	REGION 7 - Handle handshake
	    #iqUDT_HandShakeDownstreamSlip.RTS := #iqUDT_HandShakeUpstream.RTS;
	    #iqUDT_HandShakeUpstream.RTR := #iqUDT_HandShakeDownstreamSlip.RTR;
	    #iqUDT_HandShakeDownstreamSlip.TIP := #iqUDT_HandShakeUpstream.TIP;
	    #iqUDT_HandShakeDownstreamSlip.ResetEnergySave := #iqUDT_HandShakeUpstream.ResetEnergySave;
	    #iqUDT_HandShakeUpstream.CascadeStartUp := #iqUDT_HandShakeDownstreamSlip.CascadeStartUp;
	    #iqUDT_HandShakeDownstreamSlip.ReqStop := #iqUDT_HandShakeUpstream.ReqStop;
	    #iqUDT_HandShakeDownstreamSlip.DownstreamDisplacement := #iqUDT_ConveyorInterfaceDownstream.Displacement;
	END_REGION

END_FUNCTION_BLOCK

FUNCTION_BLOCK "FB_SoftVersion"
TITLE = FB_SoftVersion
{ S7_Optimized_Access := 'TRUE' }
AUTHOR : MHSE
FAMILY : GeneralSystemFunctions
VERSION : 3.0
// ATTRIBUTES
// AUTO_NUMBER = True
// BLOCK_NUMBER = 28
// END_ATTRIBUTES
//Function block to get the program checksums.
   VAR_INPUT
      is_ActualDateTime { ExternalAccessible := 'False'; ExternalVisible := 'False'; ExternalWritable := 'False'} : String;   // Actual date and time
   END_VAR

   VAR_OUTPUT
      qs_SoftVersion { ExternalAccessible := 'False'; ExternalVisible := 'False'; ExternalWritable := 'False'} : String[8];   // Software version
      qa_StandardCRC { ExternalAccessible := 'False'; ExternalVisible := 'False'; ExternalWritable := 'False'} : Array[0..7] of Byte;   // Standard program checksum output
      qa_SafetyCRC { ExternalAccessible := 'False'; ExternalVisible := 'False'; ExternalWritable := 'False'} : Array[0..7] of Byte;   // Safety program checksum output
   END_VAR

   VAR
      sFB_GetChecksum_Safety {InstructionName := 'GetChecksum'; LibVersion := '1.0'; ExternalAccessible := 'False'; ExternalVisible := 'False'; ExternalWritable := 'False'; S7_SetPoint := 'False'} : GetChecksum;   // Safety checksum read block
      sFB_GetChecksum_Standard {InstructionName := 'GetChecksum'; LibVersion := '1.0'; ExternalAccessible := 'False'; ExternalVisible := 'False'; ExternalWritable := 'False'; S7_SetPoint := 'False'} : GetChecksum;   // Standard checksum read block
   END_VAR
   VAR RETAIN
      sa_StandardCRC { ExternalAccessible := 'False'; ExternalVisible := 'False'; ExternalWritable := 'False'} : Array[0..7] of Byte;   // Standard program checksum
      sa_SafetyCRC { ExternalAccessible := 'False'; ExternalVisible := 'False'; ExternalWritable := 'False'} : Array[0..7] of Byte;   // Safety program checksum
   END_VAR
   VAR
      sa_NewStandardCRC { ExternalAccessible := 'False'; ExternalVisible := 'False'; ExternalWritable := 'False'} : Array[0..7] of Byte;   // New standard program checksum
      sa_NewSafetyCRC { ExternalAccessible := 'False'; ExternalVisible := 'False'; ExternalWritable := 'False'} : Array[0..7] of Byte;   // New safety program checksum
   END_VAR
   VAR RETAIN
      ss_Date { ExternalAccessible := 'False'; ExternalVisible := 'False'; ExternalWritable := 'False'} : String[8];   // Date charater string
   END_VAR

   VAR_TEMP
      ta_StandardCRC : Struct   // GetChecksum
         tx_Done : Bool;   // GetChecksum - Done
         tx_Busy : Bool;   // GetChecksum - Busy
         tx_Error : Bool;   // GetChecksum - Error
         tw_Status : Word;   // GetChecksum - Status
      END_STRUCT;
      ta_SafetyCRC : Struct   // GetChecksum
         tx_Done : Bool;   // GetChecksum - Done
         tx_Busy : Bool;   // GetChecksum - Busy
         tx_Error : Bool;   // GetChecksum - Error
         tw_Status : Word;   // GetChecksum - Status
      END_STRUCT;
      tx_CRCValid : Bool;   // Checksums valid
   END_VAR


BEGIN
	(*
	----------------------------------------------------------------------------------------

	Version history:
	Date        | Version   | Author        | Remark
	----------------------------------------------------------------------------------------
	24/05/2019  | 0.1       | K.Pokorski    | first release MHS TIA 15.1
	14/06/2019  | 0.2       | A.Nowak       | Replacement of instruction if for direct write into variable - Region 2
	24/07/2019  | 2.0       | L.Klar        | 2.0 MHS library release TIA 15.1
	27/08/2019  | 2.2       | K.Pokorski    | Comments adjusted
	12/11/2019  | 3.0       | P.Majka       | 3.0 MHS library release TIA 15.1
	21/02/2023  | 4.0       | F.Baten       | 4.0 Release TIA 17.5
	*)

	REGION 1 - Standard and safety program checksums

	    // Scope - 1 - Standard program CRC
	    #sFB_GetChecksum_Standard(Scope := 1,
	                              Done => #ta_StandardCRC.tx_Done,
	                              Busy => #ta_StandardCRC.tx_Busy,
	                              Error => #ta_StandardCRC.tx_Error,
	                              Status => #ta_StandardCRC.tw_Status,
	                              Checksum := #sa_NewStandardCRC);

	    // Scope - 2 - Safety program CRC
	    #sFB_GetChecksum_Safety(Scope := 2,
	                            Done => #ta_SafetyCRC.tx_Done,
	                            Busy => #ta_SafetyCRC.tx_Busy,
	                            Error => #ta_SafetyCRC.tx_Error,
	                            Status => #ta_SafetyCRC.tw_Status,
	                            Checksum := #sa_NewSafetyCRC);

	END_REGION

	REGION 2 - Checksums comparison

	    #tx_CRCValid := (#sa_NewStandardCRC = #sa_StandardCRC)
	    AND (#sa_SafetyCRC = #sa_NewSafetyCRC);

	END_REGION

	REGION 3 - New software version

	    // Separate the year, mounth and day from actual date and time and connect it to one string
	    IF (NOT #tx_CRCValid)                                           // Checksums not valid
	    THEN

	        #ss_Date := CONCAT(IN1 := MID(IN := #is_ActualDateTime,
	                                                         L := 4,
	                                                         P := 1),

	                           IN2 := MID(IN := #is_ActualDateTime,
	                                      L := 2,
	                                      P := 6),

	                           IN3 := MID(IN := #is_ActualDateTime,
	                                      L := 2,
	                                      P := 9));

	        // Standard progrm checksum update
	        #sa_StandardCRC := #sa_NewStandardCRC;

	        // Safety program checksum update
	        #sa_SafetyCRC := #sa_NewSafetyCRC;

	    END_IF;

	END_REGION

	REGION 4 - Write outputs

	    // New program date
	    #qs_SoftVersion := #ss_Date;

	    // Actual standard program checksum
	    #qa_StandardCRC := #sa_StandardCRC;

	    // Actual safety program checksum
	    #qa_SafetyCRC := #sa_SafetyCRC;

	END_REGION
END_FUNCTION_BLOCK

FUNCTION_BLOCK "FB_VfdNORDPPO4"
TITLE = Control block for NORD VFD with PPO4
{ S7_Optimized_Access := 'TRUE' }
AUTHOR : MHS
VERSION : 0.1
// ATTRIBUTES
// AUTO_NUMBER = True
// BLOCK_NUMBER = 235
// END_ATTRIBUTES
   VAR_INPUT
      iUDT_VFDConfig { ExternalAccessible := 'False'; ExternalVisible := 'False'; ExternalWritable := 'False'} : "UDT_VfdConfiguration";   // Configuration structure
      iUDT_VFDInputs { ExternalAccessible := 'False'; ExternalVisible := 'False'; ExternalWritable := 'False'} : "UDT_VfdNordPI";   // VFD inputs structure
      iUDT_MotorData { ExternalAccessible := 'False'; ExternalVisible := 'False'; ExternalWritable := 'False'} : "UDT_MotorData";   // Motor data structure
      ix_24vOk { ExternalAccessible := 'False'; ExternalVisible := 'False'; ExternalWritable := 'False'} : Bool;   // TRUE when 24VDC is healthy
      ix_400vOk { ExternalAccessible := 'False'; ExternalVisible := 'False'; ExternalWritable := 'False'} : Bool;   // TRUE when 400VAC is healthy
      ix_QuickStopDisable { ExternalAccessible := 'False'; ExternalVisible := 'False'; ExternalWritable := 'False'} : Bool := FALSE;   // TRUE when Motor can turn, False = Quick stop
      ix_SimulationModeActive { ExternalAccessible := 'False'; ExternalVisible := 'False'; ExternalWritable := 'False'} : Bool;   // TRUE when Simulation mode active
   END_VAR

   VAR_OUTPUT
      qUDT_HMIStatus { ExternalAccessible := 'False'; ExternalVisible := 'False'; ExternalWritable := 'False'} : "UDT_VfdStatus";   // HMI status structure
      qUDT_VFDOutputs { ExternalAccessible := 'False'; ExternalVisible := 'False'; ExternalWritable := 'False'} : "UDT_VfdNordPO";   // VFD outputs structure
      qUDT_commisioning { ExternalAccessible := 'False'; ExternalVisible := 'False'; ExternalWritable := 'False'} : "UDT_CommisioningNord";
   END_VAR

   VAR_IN_OUT
      iqUDT_ConveyorInterface : "UDT_ConveyorInterface";   // Conveyor interface structure
      iqUDT_VFDStatistics : "UDT_VfdStatistics";   // Satistics structure
      iqx_StartCommissioning { ExternalAccessible := 'False'; ExternalVisible := 'False'; ExternalWritable := 'False'} : Bool;   // TRUE when Start auto-commissioning
   END_VAR

   VAR
      sFB_TimerOnOffDelayCheck24V { ExternalAccessible := 'False'; ExternalVisible := 'False'; ExternalWritable := 'False'; S7_SetPoint := 'False'} : "FB_TimerOnOffDelay";   // MHS "TimerOnOffDelay" - to delay time for VFD 24V contactor
      sFB_TimerOnOffDelayCheck400V { ExternalAccessible := 'False'; ExternalVisible := 'False'; ExternalWritable := 'False'; S7_SetPoint := 'False'} : "FB_TimerOnOffDelay";   // MHS "TimerOnOffDelay" - to delay time for VFD 400V contactor
      sFB_TimerOnOffDelayVFDReset { ExternalAccessible := 'False'; ExternalVisible := 'False'; ExternalWritable := 'False'; S7_SetPoint := 'False'} : "FB_TimerOnOffDelay";   // MHS "TimerOnOffDelay" - to extend VFD reset
      sFB_TimerOnOffDelayVFDRunningFeedbackError { ExternalAccessible := 'False'; ExternalVisible := 'False'; ExternalWritable := 'False'; S7_SetPoint := 'False'} : "FB_TimerOnOffDelay";   // MHS "TimerOnOffDelay" - to delay time for VFDRunningFeedback error
      sFB_VfdNORDCommissiong { ExternalAccessible := 'False'; ExternalVisible := 'False'; ExternalWritable := 'False'; S7_SetPoint := 'False'} : "FB_VfdNORDCommissioning";   // FB to commissiong NORD drive
      sUDT_Status { ExternalAccessible := 'False'; ExternalVisible := 'False'; ExternalWritable := 'False'; S7_SetPoint := 'False'} : "UDT_VfdStatus";   // Detailed VFD status overview
      sUDT_PNDevice { ExternalAccessible := 'False'; ExternalVisible := 'False'; ExternalWritable := 'False'; S7_SetPoint := 'False'} : "UDT_PNDevice";   // PN device info structure
      sa_PNPortsStatus { ExternalAccessible := 'False'; ExternalVisible := 'False'; ExternalWritable := 'False'} : Array[1..8] of Bool;   // TRUE when specific port has an error
      sp_VFDTelegram { ExternalAccessible := 'False'; ExternalVisible := 'False'; ExternalWritable := 'False'} : HW_ANY;   // Free telegram's HW_ID
      sv_VFDGeoStruct {InstructionName := 'GEOADDR'; LibVersion := '1.0'; ExternalAccessible := 'False'; ExternalVisible := 'False'; ExternalWritable := 'False'; S7_SetPoint := 'False'} : GEOADDR;   //  Geo structure indicate to telegram
      sR_TRIG_PNSlaveNotOnline {InstructionName := 'R_TRIG'; LibVersion := '1.0'; ExternalAccessible := 'False'; ExternalVisible := 'False'; ExternalWritable := 'False'; S7_SetPoint := 'False'} : R_TRIG;   // Rising edge for trigger Profinet slave not online statistics
      sR_TRIG_PNSlaveError {InstructionName := 'R_TRIG'; LibVersion := '1.0'; ExternalAccessible := 'False'; ExternalVisible := 'False'; ExternalWritable := 'False'; S7_SetPoint := 'False'} : R_TRIG;   // Rising edge for trigger Profinet slave error statistics
      sR_TRIG_VFDInternalError {InstructionName := 'R_TRIG'; LibVersion := '1.0'; ExternalAccessible := 'False'; ExternalVisible := 'False'; ExternalWritable := 'False'; S7_SetPoint := 'False'} : R_TRIG;   // Rising edge for trigger Internal VFD Error statistics
      sR_TRIG_Running {InstructionName := 'R_TRIG'; LibVersion := '1.0'; ExternalAccessible := 'False'; ExternalVisible := 'False'; ExternalWritable := 'False'; S7_SetPoint := 'False'} : R_TRIG;   // Rising edge for starting of the running signal
      sF_TRIG_RunFwd {InstructionName := 'F_TRIG'; LibVersion := '1.0'; ExternalAccessible := 'False'; ExternalVisible := 'False'; ExternalWritable := 'False'; S7_SetPoint := 'False'} : F_TRIG;   // Falling edge for run forward signal
      sF_TRIG_RunRvs {InstructionName := 'F_TRIG'; LibVersion := '1.0'; ExternalAccessible := 'False'; ExternalVisible := 'False'; ExternalWritable := 'False'; S7_SetPoint := 'False'} : F_TRIG;   // Falling edge for run reverse signal
      sr_RPMActual { ExternalAccessible := 'False'; ExternalVisible := 'False'; ExternalWritable := 'False'} : Real;   // Drive RPM feedback
      sr_RPMSetpoint { ExternalAccessible := 'False'; ExternalVisible := 'False'; ExternalWritable := 'False'} : Real;   // Actual speed setpoint [rpm]
      sr_ReferenceFrequency { ExternalAccessible := 'False'; ExternalVisible := 'False'; ExternalWritable := 'False'} : Real;   // Frequency of the reference RPM in [Hz]
      sdi_LastRampTimeUp { ExternalAccessible := 'False'; ExternalVisible := 'False'; ExternalWritable := 'False'} : UDInt;   // Last cycle ramp down time
      sdi_LastRampTimeDown { ExternalAccessible := 'False'; ExternalVisible := 'False'; ExternalWritable := 'False'} : UDInt;   // Last cycle ramp up time
      si_ActualRamp { ExternalAccessible := 'False'; ExternalVisible := 'False'; ExternalWritable := 'False'} : UInt;   // Actual ramp value
      si_ActualRampUpTime { ExternalAccessible := 'False'; ExternalVisible := 'False'; ExternalWritable := 'False'} : UInt;   // Actual ramp up time
      si_ActualRampDownTime { ExternalAccessible := 'False'; ExternalVisible := 'False'; ExternalWritable := 'False'} : UInt;   // Actual ramp down time
      si_HWAdress { ExternalAccessible := 'False'; ExternalVisible := 'False'; ExternalWritable := 'False'} : Int;
      si_ActualSpeed { ExternalAccessible := 'False'; ExternalVisible := 'False'; ExternalWritable := 'False'} : Int;   // Actual speed in [mm/sec]
      si_Log2GeoReturn { ExternalAccessible := 'False'; ExternalVisible := 'False'; ExternalWritable := 'False'} : Int;   // Log2Geo function return
      si_Geo2LogReturn { ExternalAccessible := 'False'; ExternalVisible := 'False'; ExternalWritable := 'False'} : Int;   // Geo2Log function return
      sx_ConfigurationError { ExternalAccessible := 'False'; ExternalVisible := 'False'; ExternalWritable := 'False'} : Bool;   // Commissioning: configuration error
      sx_PNDeviceHealthy { ExternalAccessible := 'False'; ExternalVisible := 'False'; ExternalWritable := 'False'} : Bool;   // Profinet device is online and error free
      sx_HardwareAvailable { ExternalAccessible := 'False'; ExternalVisible := 'False'; ExternalWritable := 'False'} : Bool;   // Power and communication to drive are ok
      sx_VfdAvailable { ExternalAccessible := 'False'; ExternalVisible := 'False'; ExternalWritable := 'False'} : Bool;   // Hardware of VFD is ok and no communication error with movikit
      sx_24vOk { ExternalAccessible := 'False'; ExternalVisible := 'False'; ExternalWritable := 'False'} : Bool;   // 24VDC is healthy
      sx_400vOk { ExternalAccessible := 'False'; ExternalVisible := 'False'; ExternalWritable := 'False'} : Bool;   // 400VAC is healthy
      sx_ErrorActive { ExternalAccessible := 'False'; ExternalVisible := 'False'; ExternalWritable := 'False'} : Bool;   // Block has an error
      sx_EnableOperation { ExternalAccessible := 'False'; ExternalVisible := 'False'; ExternalWritable := 'False'} : Bool;   // Enable operation signal
      sx_RunVFDReverse { ExternalAccessible := 'False'; ExternalVisible := 'False'; ExternalWritable := 'False'} : Bool;   // Start VFD backward
      sx_RunVFDForward { ExternalAccessible := 'False'; ExternalVisible := 'False'; ExternalWritable := 'False'} : Bool;   // Start VFD forward
      sx_SpeedSetpointReached { ExternalAccessible := 'False'; ExternalVisible := 'False'; ExternalWritable := 'False'} : Bool;   // Motor is running at requested speed
      sx_VFDStopping { ExternalAccessible := 'False'; ExternalVisible := 'False'; ExternalWritable := 'False'} : Bool;   // VFD Stopping
      sx_VFDNotReadyError { ExternalAccessible := 'False'; ExternalVisible := 'False'; ExternalWritable := 'False'} : Bool;   // Temporary Error need to be implemented in the status
   END_VAR

   VAR CONSTANT
      cr_MaximumValueSpeedWord : Real := 16384.0;   // Maximum value of speed actual value
      cr_MaximumValueRampWord : Real := 32767.0;   // Maximum value of ramp setpoint ( corresponds to 20Sec)
      cr_MaximumFrequency : Real := 16384.0;   // Maximum value of frequency setpoint (corresponds to P105 Maximum Frequency)
      cudi_DefaultRampDownTime : UDInt := 20000;   // VFD ramp down default time [ms]
      cudi_DefaultRampUpTime : UDInt := 20000;   // VFD ramp up default time [ms]
      ci_VFDArea : UInt := 1;   // Area ID of IO Profinet devices
      ci_SubmoduleHWType : UInt := 5;   // Submodule HW_type number
      ci_TelegramSlot : UInt := 0;   // PPO4 telegram slot
      ci_TelegramSubslot : UInt := 1;   // PPO4 telegram subslot
      ci_NumberOfProfinetPorts : Int := 2;   // Number of Profinet ports in device
   END_VAR


BEGIN
	(*
	----------------------------------------------------------------------------------------

	Version history:
	Date        | Version   | Author        | Remark
	----------------------------------------------------------------------------------------
	25/01/2020  | 0.1       | S.Theocharis  | Initial version TIA 15.1
	28/04/2022  | 0.2       | K. Pokorski   | NORD Commissioning interface change
	09/05/2022  | 0.3       | M. Pluskota   | Reference speed changed to nominal speed for actual speed calculation
	12/05/2022  | 0.4       | M. Pluskota   | Ramp equation adjustet for nord drives
	04/06/2022  | 0.5       | M. Pluskota   | Aded a if statment to not exceed the max value of the ramp value
	                                        | Error decoding changed now the error is shown as ErrorCode.SubErrorCodee
	12/07/2022  | 0.6       | M. Pluskota   | Ramp equation bug fix
	29/07/2022  | 0.7       | M. Piela      | Add hardware ok to the profinet checking
	21/02/2023  | 4.0       | F.Baten       | 4.0 Release TIA 17.5
	*)


	REGION 1 - Get Device Profinet information

	    "FC_GetDevicePN"(is_PNDeviceName := #iUDT_VFDConfig.VFDPNDeviceName,
	                     ix_SimulationModeActive := #ix_SimulationModeActive,
	                     iqUDT_PND := #sUDT_PNDevice);


	    "FC_GetPNPortStatus"(ii_NumberOfPorts := #ci_NumberOfProfinetPorts,
	                         iUDT_DevicePNInfo := #sUDT_PNDevice,
	                         qa_PortFault => #sa_PNPortsStatus);

	END_REGION

	REGION 2 - Reset errors

	    IF #iqUDT_ConveyorInterface.InternalErrorReset OR (NOT #iqUDT_ConveyorInterface.HardwareOk AND #sUDT_Status.PNSlaveNotonline)   // Reser errors when Reset is given
	    THEN

	        #sUDT_Status.PNSlaveNotonline := FALSE;
	        #sUDT_Status.PNSlaveError := FALSE;
	        #sUDT_Status.InternalError := FALSE;
	        #sUDT_Status.VFDRunningFeedbackError := FALSE;
	        #sUDT_Status.PNSlaveWarning := FALSE;

	    END_IF;


	    // Create  extended pulse for VFD Reset
	    #sFB_TimerOnOffDelayVFDReset(iudi_OnDelayTime := 0,
	                                 iudi_OffDelayTime := 200,
	                                 ix_SignalToDelay := #iqUDT_ConveyorInterface.InternalErrorReset,
	                                 ix_Enable := TRUE);

	END_REGION

	REGION 3 - Hardware checks
	    // Hardware will only be available after the delay, so the device has time for the initialisation
	    #sFB_TimerOnOffDelayCheck24V(iudi_OnDelayTime := 2000,
	                                 iudi_OffDelayTime := 0,
	                                 ix_SignalToDelay := #ix_24vOk
	    );

	    #sx_24vOk := #sFB_TimerOnOffDelayCheck24V.qx_DelayedSignal;

	    #sFB_TimerOnOffDelayCheck400V(iudi_OnDelayTime := 2000,
	                                  ix_SignalToDelay := #ix_400vOk);

	    #sx_400vOk := #sFB_TimerOnOffDelayCheck400V.qx_DelayedSignal;

	    // Check if PN device is online
	    IF NOT "DB_ProfinetDiagnostic".ProfinetNetworks[#sUDT_PNDevice.PNNetworknumber].DeviceStatus[#sUDT_PNDevice.PNDeviceNumber].DeviceState.Exist
	        AND NOT #ix_SimulationModeActive
	        AND #sx_24vOk
	        AND #iqUDT_ConveyorInterface.HardwareOk
	    THEN
	        #sUDT_Status.PNSlaveNotonline := TRUE;

	    END_IF;

	    // Check if PN ports are healthy
	    IF #sa_PNPortsStatus[1] XOR #sa_PNPortsStatus[2] THEN
	        #sUDT_Status.PNSlaveWarning := TRUE;
	    END_IF;


	    // Check if PN device has an error
	    IF "DB_ProfinetDiagnostic".ProfinetNetworks[#sUDT_PNDevice.PNNetworknumber].DeviceStatus[#sUDT_PNDevice.PNDeviceNumber].DeviceState.Error
	        AND NOT #ix_SimulationModeActive
	        AND #sx_24vOk
	        AND NOT #sUDT_Status.PNSlaveWarning
	        AND #iqUDT_ConveyorInterface.HardwareOk
	    THEN
	        #sUDT_Status.PNSlaveError := TRUE;
	    END_IF;

	    // Set bit when PN device is healthy (online and no error)
	    #sx_PNDeviceHealthy := NOT #sUDT_Status.PNSlaveNotonline
	    AND NOT #sUDT_Status.PNSlaveError
	    AND #sUDT_PNDevice.PNDeviceFound
	    AND #sx_24vOk;

	    // Set hardware available bit when all conditions are met
	    #sx_HardwareAvailable := (#sx_24vOk
	    AND #sx_PNDeviceHealthy)
	    OR #ix_SimulationModeActive;


	    // VFD is ready for operation if hardware ok
	    #sx_VfdAvailable := #sx_HardwareAvailable;

	    //VFD not ready error . Temporary
	    #sx_VFDNotReadyError := #sx_HardwareAvailable
	    AND NOT #iUDT_VFDInputs.ZSW.ReadyToStart
	    AND #iUDT_VFDInputs.ZSW.EmergencyStop
	    OR NOT #iUDT_VFDInputs.ZSW.BusControlActive;




	END_REGION

	REGION 4 - Check errors and warnings

	    // Check if the VFD has a warning
	    #sUDT_Status.InternalWarning := #iUDT_VFDInputs.ZSW.WarningActive;

	    // Copy warning code to status DB when warning active
	    IF #sUDT_Status.InternalWarning
	    THEN

	        #sUDT_Status.ErrorCode := #iUDT_VFDInputs.FaultCode / 10; // AST check the value of warning
	        #sUDT_Status.SubErrorCode := #iUDT_VFDInputs.FaultCode MOD 10;

	    END_IF;

	    // Check if the VFD has an error
	    #sUDT_Status.InternalError := #iUDT_VFDInputs.ZSW.Fault; // AND NOT #sx_StartMeasuring;

	    // Copy error code to status DB when error active
	    IF #sUDT_Status.InternalError
	    THEN

	        #sUDT_Status.ErrorCode := #iUDT_VFDInputs.FaultCode / 10; // AST check the value of warning
	        #sUDT_Status.SubErrorCode := #iUDT_VFDInputs.FaultCode MOD 10;

	    END_IF;

	    // Reset error code if warning and error not available
	    IF (NOT #sUDT_Status.InternalWarning
	        AND NOT #sUDT_Status.InternalError)
	    THEN

	        #sUDT_Status.ErrorCode := 0;
	        #sUDT_Status.SubErrorCode := 0;
	    END_IF;

	END_REGION

	REGION 5 - Check if configuration is ok for commissioning purposes

	    IF #iUDT_VFDConfig.WheelEndPerimeter > 0.0                                         // If perimeter of wheel at the end of gear is greater than 0
	        AND #iUDT_VFDConfig.GearRatio > 0.0                                            // and gear ratio is greater than 0
	        AND #iUDT_VFDConfig.ReferenceRPM > 0.0                                         // and maximum speed is greater than 0
	        AND #iUDT_VFDConfig.VFDRampUpTime > 0                                          // and ramp up time is greater than 0
	        AND #iUDT_VFDConfig.VFDRampDownTime > 0                                        // and ramp down time is greater than zero
	        AND #iUDT_VFDConfig.VFDStartupTime > 0.0                                       // and startup time is greater then zero
	        //  AND MOTOR NOMINAL SPEED IS >0  the reference speed is invalid for NORD drives
	        AND #cudi_DefaultRampUpTime > #iUDT_VFDConfig.VFDRampUpTime                     // and ramp up time is not greater than default ramp up time
	        AND #cudi_DefaultRampDownTime > #iUDT_VFDConfig.VFDRampDownTime                 // and ramp down time is not greater than default ramp down time
	        // need to know if the FI receives a percentage of a default ramp or value in ms , depending to that the configuration validation code will change

	        AND (#sUDT_PNDevice.PNDeviceFound                                              // and device not found in PN structure
	        OR #ix_SimulationModeActive)                                                    // or simulation mode is active
	    THEN
	        #sx_ConfigurationError := FALSE;                                                // Reset configuration error
	    ELSE
	        #sx_ConfigurationError := TRUE;                                                 // Set configuration error
	    END_IF;
	    #qUDT_commisioning.CommissionError := #sx_ConfigurationError;

	END_REGION

	REGION 6 - Speed handling

	    //Calculate actual speed value in rpm
	    // #sr_RPMActual := ((INT_TO_REAL(#i_UDT_VFDInputs.ActualSpeed) / #cr_MaximumValueSpeedWord) * INT_TO_REAL(#i_UDT_MotorData.NominalSpeed));

	    //#sr_RPMActual := ((INT_TO_REAL(#i_UDT_VFDInputs.ActualSpeed) / #cr_MaximumValueSpeedWord) * (#i_UDT_MotorData.NominalSpeed));
	    #sr_RPMActual := ((INT_TO_REAL(#iUDT_VFDInputs.ActualSpeed) / #cr_MaximumFrequency) * (#iUDT_VFDConfig.ReferenceRPM));
	    // Calculate actual speed in mm/s
	    #si_ActualSpeed := REAL_TO_INT((#sr_RPMActual / #iUDT_VFDConfig.GearRatio) * ((#iUDT_VFDConfig.WheelEndPerimeter) / 60.0));


	    //change the i_UDT_VFDInput.Actualspeed to RPM

	    // Reversal actual speed
	    IF #iUDT_VFDConfig.DirectionReversal THEN

	        #si_ActualSpeed := #si_ActualSpeed * -1;

	    END_IF;

	    // Calculate actual speed setpoint in rpm
	    #sr_RPMSetpoint := ((DINT_TO_REAL(INT_TO_DINT(#iqUDT_ConveyorInterface.SpeedSetpoint) * 60)) / #iUDT_VFDConfig.WheelEndPerimeter) * #iUDT_VFDConfig.GearRatio;

	    // Check if speed setpoint is reached
	    #sx_SpeedSetpointReached := (ABS(#si_ActualSpeed) >= (#iqUDT_ConveyorInterface.SpeedSetpoint - #iUDT_VFDConfig.SpeedSetpointWindow))
	    AND (ABS(#si_ActualSpeed) <= (#iqUDT_ConveyorInterface.SpeedSetpoint + #iUDT_VFDConfig.SpeedSetpointWindow));


	END_REGION

	REGION 7 - Prepare output data VFD

	    REGION 7.1 - Set speed setpoint in forward and reverse directory

	        // If motor stopped and Run forward is requested and interlock forward is active, the speed setpoint is loaded to run forward.
	        //  IF (#i_UDT_VFDInputs.ActualSpeed = 0) AND #iq_UDT_ConveyorInterface.RunFwd AND #i_UDT_VFDConfig.InterlockFwd
	        IF #iqUDT_ConveyorInterface.RunFwd AND #iUDT_VFDConfig.InterlockFwd
	        THEN
	            #sx_RunVFDForward := TRUE;
	            #sx_RunVFDReverse := FALSE;
	        END_IF;

	        // If motor stopped and Run reverse is requested and interlock reverse is active, the speed setpoint is loaded to run reverse.
	        IF (#iUDT_VFDInputs.ActualSpeed = 0) AND #iqUDT_ConveyorInterface.RunRvs AND #iUDT_VFDConfig.InterlockRvs
	        THEN
	            #sx_RunVFDReverse := TRUE;
	            #sx_RunVFDForward := FALSE;
	        END_IF;

	    END_REGION

	    REGION 7.2 - Stopping

	        // Create trigger when direction signal falling
	        #sF_TRIG_RunFwd(CLK := #iqUDT_ConveyorInterface.RunFwd);
	        #sF_TRIG_RunRvs(CLK := #iqUDT_ConveyorInterface.RunRvs);

	        // When no run signal is given the VFD should stop
	        IF NOT #iqUDT_ConveyorInterface.RunRvs AND NOT #iqUDT_ConveyorInterface.RunFwd
	            OR (#iqUDT_ConveyorInterface.RunRvs AND #iqUDT_ConveyorInterface.RunFwd)
	            OR #sF_TRIG_RunRvs.Q
	            OR #sF_TRIG_RunFwd.Q

	        THEN
	            #sx_RunVFDReverse := FALSE;
	            #sx_RunVFDForward := FALSE;
	        END_IF;

	        IF NOT #sx_RunVFDReverse AND NOT #sx_RunVFDForward AND (#iUDT_VFDInputs.ActualSpeed <> 0)
	        THEN
	            #sx_VFDStopping := TRUE;
	        ELSE
	            #sx_VFDStopping := FALSE;
	        END_IF;

	    END_REGION

	    REGION 7.3 - Check for enable operation signal

	        #sx_EnableOperation := #sx_VfdAvailable
	        AND #sx_400vOk
	        AND NOT #sx_ConfigurationError
	        AND (#sx_RunVFDForward OR #sx_RunVFDReverse); // add communication error

	    END_REGION

	    REGION 7.4 - Write acceleration and deceleration value to drive

	        //Detect is VFD is ramping up
	        IF ABS(#sr_RPMSetpoint) > ABS(#sr_RPMActual)
	            AND NOT #sx_SpeedSetpointReached
	            AND #iUDT_VFDInputs.ZSW.OperationEnabled
	            AND (#sx_RunVFDForward OR #sx_RunVFDReverse)
	        THEN
	            // Calculate the ramp up time if the vfd configuration is changed durning process or the vfd starts from speed 0
	            IF #sdi_LastRampTimeUp <> #iUDT_VFDConfig.VFDRampUpTime THEN
	                #si_ActualRamp := REAL_TO_UINT(UDINT_TO_REAL(#iUDT_VFDConfig.VFDRampUpTime) / UDINT_TO_REAL(#cudi_DefaultRampUpTime) * #cr_MaximumValueRampWord / (#sr_RPMSetpoint / #iUDT_VFDConfig.ReferenceRPM));
	                #si_ActualRampUpTime := #si_ActualRamp;
	            ELSE
	                #si_ActualRamp := #si_ActualRampUpTime;
	            END_IF;
	            #sdi_LastRampTimeUp := #iUDT_VFDConfig.VFDRampUpTime;
	        ELSE
	            // Calculate the ramp down time if the actual speed is greater than 0 and the configuration has changed durning process
	            // or the VFD perform the first deceleration

	            IF #si_ActualSpeed <> 0 THEN
	                IF #sdi_LastRampTimeDown <> #iUDT_VFDConfig.VFDRampDownTime
	                THEN
	                    #si_ActualRamp := REAL_TO_UINT(UDINT_TO_REAL(#iUDT_VFDConfig.VFDRampDownTime) / UDINT_TO_REAL(#cudi_DefaultRampDownTime) * #cr_MaximumValueRampWord / (#sr_RPMSetpoint / #iUDT_VFDConfig.ReferenceRPM));
	                    #si_ActualRampDownTime := #si_ActualRamp;

	                ELSE
	                    #si_ActualRamp := #si_ActualRampDownTime;
	                END_IF;
	                #sdi_LastRampTimeDown := #iUDT_VFDConfig.VFDRampDownTime;
	            ELSE
	                #sdi_LastRampTimeDown := 0;
	                #sdi_LastRampTimeUp := 0;
	            END_IF;

	        END_IF;

	        // If the ramp value exceeds the maximum value, then the maximum value is sent to the VFD
	        IF UINT_TO_REAL(#si_ActualRamp) > #cr_MaximumValueRampWord
	        THEN
	            #qUDT_VFDOutputs.RampTimeSetPoint := REAL_TO_INT(#cr_MaximumValueRampWord);
	        ELSE
	            #qUDT_VFDOutputs.RampTimeSetPoint := REAL_TO_INT(UINT_TO_REAL(#si_ActualRamp));
	        END_IF;


	    END_REGION
	END_REGION

	REGION 8 - Auto Commmissioning

	    REGION 8.1 Initialize
	        IF #iqx_StartCommissioning THEN

	            //Caclulate theoretical reference Hz. Necessary for NORD drives cause the setpoint is given at Hz
	            //Variation of motor slip from 50Hz to reference Hz is not taken into account. That means there will always be a variantion between Setpoint and actual speed
	            #sr_ReferenceFrequency := (#iUDT_VFDConfig.ReferenceRPM / 1500) * 50; //1500 for 4 pole motor

	            // Get hardware adres of "SK-TU4-PNS~Head" submodule
	            #si_Log2GeoReturn := LOG2GEO(LADDR := "DB_ProfinetDiagnostic".ProfinetNetworks[#sUDT_PNDevice.PNNetworknumber].DeviceStatus[#sUDT_PNDevice.PNDeviceNumber].DeviceState.HW_ID, GEOADDR := #sv_VFDGeoStruct);       // "LOG2GEO" to get profinet network number
	            #sv_VFDGeoStruct.AREA := #ci_VFDArea;                                                                                                                                                                               // Set IO Profinet devices area ID
	            #sv_VFDGeoStruct.HWTYPE := #ci_SubmoduleHWType;                                                                                                                                                                     // Set submodule HW_type number
	            #sv_VFDGeoStruct.STATION := INT_TO_UINT(#sUDT_PNDevice.PNDeviceNumber);                                                                                                                                            // Set device's profinet number
	            #sv_VFDGeoStruct.SLOT := #ci_TelegramSlot;                                                                                                                                                                          // Set free telegram slot
	            #sv_VFDGeoStruct.SUBSLOT := #ci_TelegramSubslot;                                                                                                                                                                    // Set free telegram subslot

	            #si_Geo2LogReturn := GEO2LOG(GEOADDR := #sv_VFDGeoStruct, LADDR => #sp_VFDTelegram);                                                                                                                              // "GEO2LOG" to get free telegram's HW_ID

	        END_IF;

	    END_REGION

	    REGION 8.2 Run - auto commissioning

	        #sFB_VfdNORDCommissiong(ix_VFDReadyToRun := #sx_400vOk AND #iUDT_VFDInputs.ZSW.EmergencyStop AND NOT #iUDT_VFDInputs.ZSW.Fault,
	                                qx_24VCommissioningDone => #sFB_VfdNORDCommissiong.qx_24VCommissioningDone,
	                                iqx_Enable := #iqx_StartCommissioning,
	                                ir_ReferenceFrequency := #sr_ReferenceFrequency,
	                                ihw_HardwareID := #sp_VFDTelegram,
	                                iudt_MotorData := #iUDT_MotorData,
	                                qi_HWAdress => #qUDT_commisioning.HWAdress,
	                                qx_Busy => #sFB_VfdNORDCommissiong.qx_Busy,
	                                qx_Done => #sFB_VfdNORDCommissiong.qx_Done,
	                                qx_Error => #sFB_VfdNORDCommissiong.qx_Error);

	    END_REGION

	END_REGION

	REGION 9 - Write outputs to VFD

	    REGION 9.1 - Write control word 1

	        #qUDT_VFDOutputs.STW.ReadyForOperation := #sx_RunVFDReverse OR #sx_RunVFDForward;
	        #qUDT_VFDOutputs.STW.DisableVoltage := TRUE;
	        #qUDT_VFDOutputs.STW.EmergencyStop := #ix_QuickStopDisable;
	        #qUDT_VFDOutputs.STW.EnableOperation := TRUE;
	        #qUDT_VFDOutputs.STW.EnablePulsles := TRUE;
	        #qUDT_VFDOutputs.STW.EnableRamp := TRUE;
	        #qUDT_VFDOutputs.STW.EnableSetpoint := TRUE;
	        #qUDT_VFDOutputs.STW.Acknowledge := #sFB_TimerOnOffDelayVFDReset.qx_DelayedSignal;
	        #qUDT_VFDOutputs.STW."StartFunction408.11" := FALSE;
	        #qUDT_VFDOutputs.STW."StartFunction408.12" := FALSE;
	        #qUDT_VFDOutputs.STW.ControlDataValid := TRUE;
	        #qUDT_VFDOutputs.STW.RotationRightOn := TRUE; //direction reversal via the speed setpoint
	        #qUDT_VFDOutputs.STW.RotationLeftOn := FALSE;
	        #qUDT_VFDOutputs.STW.Reserved := FALSE;
	        #qUDT_VFDOutputs.STW.ParameterSetBit0 := FALSE; //Parameter set 1
	        #qUDT_VFDOutputs.STW.ParameterSetBit1 := FALSE; //Parameter set 1

	        IF (NOT #sx_VfdAvailable OR NOT #sx_400vOk) //AND NOT #sx_StartMeasuring
	        THEN
	            #qUDT_VFDOutputs.STW.ReadyForOperation := FALSE;
	            #qUDT_VFDOutputs.STW.EmergencyStop := FALSE;
	            #qUDT_VFDOutputs.STW.EnableSetpoint := FALSE;
	            #qUDT_VFDOutputs.STW."StartFunction408.11" := FALSE;
	            #qUDT_VFDOutputs.STW."StartFunction408.12" := FALSE;
	        END_IF;
	    END_REGION

	    REGION 9.2 - Write speed setpoint to drive

	        // Calculate normalized speed setpoint
	        #qUDT_VFDOutputs.FrequencySetPoint := REAL_TO_INT((#sr_RPMSetpoint / #iUDT_VFDConfig.ReferenceRPM) * #cr_MaximumFrequency);

	        IF #qUDT_VFDOutputs.FrequencySetPoint > #cr_MaximumFrequency
	        THEN
	            #qUDT_VFDOutputs.FrequencySetPoint := REAL_TO_INT(#cr_MaximumFrequency);
	        END_IF;

	        // The conveyor stopped and may now run in reverse direction
	        IF (#sx_RunVFDReverse AND NOT #iUDT_VFDConfig.DirectionReversal)
	            OR (#sx_RunVFDForward AND #iUDT_VFDConfig.DirectionReversal)
	        THEN
	            #qUDT_VFDOutputs.FrequencySetPoint := #qUDT_VFDOutputs.FrequencySetPoint * -1;
	        END_IF;

	        // Clear speed setpoint when no run request or above direction request or is configuration error
	        IF (NOT #sx_RunVFDForward AND NOT #sx_RunVFDReverse)
	            OR #sx_ConfigurationError
	        THEN
	            #qUDT_VFDOutputs.FrequencySetPoint := 0;
	        END_IF;

	    END_REGION

	END_REGION

	REGION 10 - Check if motor is running

	    //The motor should start running after specific time. If not the VFDRunningFeedback error occured
	    #sFB_TimerOnOffDelayVFDRunningFeedbackError(iudi_OnDelayTime := #iUDT_VFDConfig.VFDStartupTime,
	                                                ix_SignalToDelay := #sx_EnableOperation AND NOT (#si_ActualSpeed <> 0));

	    IF #sFB_TimerOnOffDelayVFDRunningFeedbackError.qx_DelayedSignal THEN

	        #sUDT_Status.VFDRunningFeedbackError := TRUE;

	    END_IF;



	END_REGION

	REGION 11 - Copy signals to interface DB and to status output UDT

	    // Create internal error status
	    #sx_ErrorActive := #sUDT_Status.PNSlaveNotonline
	    OR #sUDT_Status.VFDRunningFeedbackError
	    OR #sUDT_Status.PNSlaveError //Commented out BY AST TO allow run in ring topology v3.12
	    OR #sUDT_Status.InternalError;

	    // Write interface bits - AST Check thoses statuses
	    #iqUDT_ConveyorInterface.VFDRunning := #sx_VfdAvailable AND (#iqUDT_ConveyorInterface.ActualSpeed <> 0 OR #qUDT_VFDOutputs.STW.ReadyForOperation);   // Write true on output Conveyor interface structure if VFD is in operation and motor is turning
	    #iqUDT_ConveyorInterface.VFDatSpeed := #sx_SpeedSetpointReached AND #sx_VfdAvailable AND #si_ActualSpeed <> 0;                                                                                                  // Copy setpoint speed reached state from static to the output conveyor interface structure
	    #iqUDT_ConveyorInterface.InternalWarningVFD := #iUDT_VFDInputs.ZSW.WarningActive;                                                                                                      // Set the internal VFD warning bit if any warning is active
	    #iqUDT_ConveyorInterface.InternalErrorVFD := #sx_ErrorActive;                                                                                                                           // Set the internal VFD error bit if any fault is active
	    #iqUDT_ConveyorInterface.ActualSpeed := #si_ActualSpeed;                                                                                                                                // Copy the calculated value to the output
	    #iqUDT_ConveyorInterface.ConfigurationError := #iqUDT_ConveyorInterface.ConfigurationError OR #sx_ConfigurationError;

	    // Copy error status to output
	    #qUDT_HMIStatus := #sUDT_Status;

	END_REGION

	REGION 12 - Statistic
	    // Create trigger on error and create statistics for profinet slave not online
	    #sR_TRIG_PNSlaveNotOnline(CLK := #sUDT_Status.PNSlaveNotonline);                                        // Detect the rising edge of the error

	    IF #iqUDT_ConveyorInterface.ResetStatistics OR #sUDT_Status.PNSlaveNotonline
	    THEN

	        "FC_Statistics"(ix_Reset := #iqUDT_ConveyorInterface.ResetStatistics,
	                        ix_Activate := #sUDT_Status.PNSlaveNotonline,
	                        ix_RTrigActivate := #sR_TRIG_PNSlaveNotOnline.Q,
	                        iqUDT_Statistics := #iqUDT_VFDStatistics.PNSlaveNotOnline);
	    END_IF;

	    // Create trigger on error and create statistics for profinet slave error
	    #sR_TRIG_PNSlaveError(CLK := #sUDT_Status.PNSlaveError);                                        // Detect the rising edge of the error

	    IF #iqUDT_ConveyorInterface.ResetStatistics OR #sUDT_Status.PNSlaveError
	    THEN

	        "FC_Statistics"(ix_Reset := #iqUDT_ConveyorInterface.ResetStatistics,
	                        ix_Activate := #sUDT_Status.PNSlaveError,
	                        ix_RTrigActivate := #sR_TRIG_PNSlaveError.Q,
	                        iqUDT_Statistics := #iqUDT_VFDStatistics.PNSlaveError);
	    END_IF;

	    // Create trigger on error and create statistics for internal VFD Error
	    #sR_TRIG_VFDInternalError(CLK := #sUDT_Status.InternalError);                                        // Detect the rising edge of the error

	    IF #iqUDT_ConveyorInterface.ResetStatistics OR #sUDT_Status.InternalError
	    THEN

	        "FC_Statistics"(ix_Reset := #iqUDT_ConveyorInterface.ResetStatistics,
	                        ix_Activate := #sUDT_Status.InternalError,
	                        ix_RTrigActivate := #sR_TRIG_VFDInternalError.Q,
	                        iqUDT_Statistics := #iqUDT_VFDStatistics.VFDInternalError);
	    END_IF;

	    // Create trigger on running signal and create statistics for running status
	    #sR_TRIG_Running(CLK := #iqUDT_ConveyorInterface.VFDRunning);                                        // Detect the rising edge of the signal

	    IF #iqUDT_ConveyorInterface.ResetStatistics OR #iqUDT_ConveyorInterface.VFDRunning
	    THEN

	        "FC_Statistics"(ix_Reset := #iqUDT_ConveyorInterface.ResetStatistics,
	                        ix_Activate := #iqUDT_ConveyorInterface.VFDRunning,
	                        ix_RTrigActivate := #sR_TRIG_Running.Q,
	                        iqUDT_Statistics := #iqUDT_VFDStatistics.Running);
	    END_IF;

	END_REGION
END_FUNCTION_BLOCK

FUNCTION_BLOCK "FB_SystemStatistics"
{ S7_Optimized_Access := 'TRUE' }
AUTHOR : MHS
VERSION : 3.0
// ATTRIBUTES
// AUTO_NUMBER = True
// BLOCK_NUMBER = 29
// END_ATTRIBUTES
   VAR_INPUT
      ix_HMIStop { ExternalAccessible := 'False'; ExternalVisible := 'False'; ExternalWritable := 'False'} : Bool;   // HMI stop button one shot signal
      ix_FieldStop { ExternalAccessible := 'False'; ExternalVisible := 'False'; ExternalWritable := 'False'} : Bool;   // Field stop button one shot signal
      ix_BuildingEStop { ExternalAccessible := 'False'; ExternalVisible := 'False'; ExternalWritable := 'False'} : Bool;   // TRUE if bulding emergency stop button is active
      ix_MCPEStop { ExternalAccessible := 'False'; ExternalVisible := 'False'; ExternalWritable := 'False'} : Bool;   // TRUE if MCP emergency stop button is active
      ix_RemotePanelEStop { ExternalAccessible := 'False'; ExternalVisible := 'False'; ExternalWritable := 'False'} : Bool;   // TRUE if Remote Panel emergency stop button is active
   END_VAR

   VAR_IN_OUT
      iqUDT_EquipmentControl : "UDT_EquipmentControl";   // Equipment control structure
      iqUDT_Statistics : "UDT_SystemStatistics";   // Statistics structure
   END_VAR

   VAR
      sR_Trig_HMIStop {InstructionName := 'R_TRIG'; LibVersion := '1.0'; ExternalAccessible := 'False'; ExternalVisible := 'False'; ExternalWritable := 'False'; S7_SetPoint := 'False'} : R_TRIG;   // Rise trigger when a HMI stop is active
      sR_Trig_FieldStop {InstructionName := 'R_TRIG'; LibVersion := '1.0'; ExternalAccessible := 'False'; ExternalVisible := 'False'; ExternalWritable := 'False'; S7_SetPoint := 'False'} : R_TRIG;   // Rise trigger when a field stop is active
      sR_Trig_BuildingEStop {InstructionName := 'R_TRIG'; LibVersion := '1.0'; ExternalAccessible := 'False'; ExternalVisible := 'False'; ExternalWritable := 'False'; S7_SetPoint := 'False'} : R_TRIG;   // Rise trigger when a building emergency stop is active
      sR_Trig_MCPEStop {InstructionName := 'R_TRIG'; LibVersion := '1.0'; ExternalAccessible := 'False'; ExternalVisible := 'False'; ExternalWritable := 'False'; S7_SetPoint := 'False'} : R_TRIG;   // Rise trigger when a MCP emergency stop is active
      sR_Trig_RemotePanelEStop {InstructionName := 'R_TRIG'; LibVersion := '1.0'; ExternalAccessible := 'False'; ExternalVisible := 'False'; ExternalWritable := 'False'; S7_SetPoint := 'False'} : R_TRIG;   // Rise trigger when a remote panel emergency stop is active
      sR_TRIG_AutomaticOn {InstructionName := 'R_TRIG'; LibVersion := '1.0'; ExternalAccessible := 'False'; ExternalVisible := 'False'; ExternalWritable := 'False'; S7_SetPoint := 'False'} : R_TRIG;   // Rise trigger when a automatic mode  is active
      sR_TRIG_DataReset {InstructionName := 'R_TRIG'; LibVersion := '1.0'; ExternalAccessible := 'False'; ExternalVisible := 'False'; ExternalWritable := 'False'; S7_SetPoint := 'False'} : R_TRIG;   // Rise trigger when data reset command is received
      sR_TRIG_Error {InstructionName := 'R_TRIG'; LibVersion := '1.0'; ExternalAccessible := 'False'; ExternalVisible := 'False'; ExternalWritable := 'False'; S7_SetPoint := 'False'} : R_TRIG;   // Rise trigger when  Error occured
      sF_TRIG_Error {InstructionName := 'F_TRIG'; LibVersion := '1.0'; ExternalAccessible := 'False'; ExternalVisible := 'False'; ExternalWritable := 'False'; S7_SetPoint := 'False'} : F_TRIG;   // Fall trigger when  Error is cleared
      sx_HMIStop { ExternalAccessible := 'False'; ExternalVisible := 'False'; ExternalWritable := 'False'} : Bool;   // HMI stop signal
      sx_FieldStop { ExternalAccessible := 'False'; ExternalVisible := 'False'; ExternalWritable := 'False'} : Bool;   // Field stop signal
   END_VAR


BEGIN
	(*
	----------------------------------------------------------------------------------------

	Version history:
	Date        | Version   | Author        | Remark
	----------------------------------------------------------------------------------------
	14/01/2020  | 3.0       | S. Nikodem    | first release MHS TIA 15.1
	22/08/2020  | 3.1       | S. Theocharis | Updated for UPS EMA HMI
	03/08/2021  | 3.2       | M. Roijen     | Bug fix System in error iq_UDT_Statistics
	21/02/2023  | 4.0       | F.Baten       | 4.0 Release TIA 17.5
	*)

	REGION 1 – Triggers

	    // Rise trigger when a HMI stop is active
	    #sR_Trig_HMIStop(CLK := #sx_HMIStop);

	    // Rise trigger when a field stop is active
	    #sR_Trig_FieldStop(CLK := #sx_FieldStop);

	    // Rise trigger when a building emergency stop is active trigger
	    #sR_Trig_BuildingEStop(CLK := #ix_BuildingEStop);

	    // Rise trigger when a MCP emergency stop is active
	    #sR_Trig_MCPEStop(CLK := #ix_MCPEStop);

	    // Rise trigger when a remote panel emergency stop is active
	    #sR_Trig_RemotePanelEStop(CLK := #ix_RemotePanelEStop);

	    // Rise trigger when a Field stop is active
	    #sR_TRIG_AutomaticOn(CLK := #iqUDT_EquipmentControl.Command.AutomaticOn);

	    // Fall trigger when error is cleared (UPS EMA Addition)
	    #sF_TRIG_Error(CLK := #iqUDT_EquipmentControl.Report.Error);

	    //Rise trigger when data reset command is received (UPS EMA Addition)
	    #sR_TRIG_DataReset(CLK := #iqUDT_EquipmentControl.Command.ResetData);

	    //Rise trigger on error
	    #sR_TRIG_Error(CLK := #iqUDT_EquipmentControl.Report.Error);

	END_REGION

	REGION 2 – Sustain input signals

	    // Set HMI stop when input signal and automatic mode are active
	    IF #ix_HMIStop AND #iqUDT_EquipmentControl.Command.AutomaticOn THEN

	        #sx_HMIStop := TRUE;

	    END_IF;

	    // Set Field stop when input signal and automatic mode are active
	    IF #ix_FieldStop AND #iqUDT_EquipmentControl.Command.AutomaticOn THEN

	        #sx_FieldStop := TRUE;

	    END_IF;

	    /// Reset when automatic mode is active
	    IF #sR_TRIG_AutomaticOn.Q THEN

	        #sx_HMIStop := FALSE;
	        #sx_FieldStop := FALSE;

	    END_IF;
	END_REGION

	REGION 3 – Statistics

	    // HMI stop signal statistics
	    IF #sx_HMIStop
	        OR #iqUDT_EquipmentControl.Command.ResetData
	    THEN

	        "FC_Statistics"(ix_Reset := #iqUDT_EquipmentControl.Command.ResetData,
	                        ix_Activate := #sx_HMIStop,
	                        ix_RTrigActivate := #sR_Trig_HMIStop.Q,
	                        iqUDT_Statistics := #iqUDT_Statistics.HMI_Stop);
	    END_IF;

	    // Field stop signal statistics
	    IF #sx_FieldStop
	        OR #iqUDT_EquipmentControl.Command.ResetData
	    THEN

	        "FC_Statistics"(ix_Reset := #iqUDT_EquipmentControl.Command.ResetData,
	                        ix_Activate := #sx_FieldStop,
	                        ix_RTrigActivate := #sR_Trig_FieldStop.Q,
	                        iqUDT_Statistics := #iqUDT_Statistics."Field_Stop");
	    END_IF;

	    // Building emergency stop statistics
	    IF #ix_BuildingEStop
	        OR #iqUDT_EquipmentControl.Command.ResetData
	    THEN

	        "FC_Statistics"(ix_Reset := #iqUDT_EquipmentControl.Command.ResetData,
	                        ix_Activate := #ix_BuildingEStop,
	                        ix_RTrigActivate := #sR_Trig_BuildingEStop.Q,
	                        iqUDT_Statistics := #iqUDT_Statistics."Building_EStop");
	    END_IF;


	    // MCP emergency stop statistics
	    IF #ix_MCPEStop
	        OR #iqUDT_EquipmentControl.Command.ResetData
	    THEN

	        "FC_Statistics"(ix_Reset := #iqUDT_EquipmentControl.Command.ResetData,
	                        ix_Activate := #ix_MCPEStop,
	                        ix_RTrigActivate := #sR_Trig_MCPEStop.Q,
	                        iqUDT_Statistics := #iqUDT_Statistics."MCP_EStop");

	    END_IF;

	    // Remote panel emergency stop statistics
	    IF #ix_RemotePanelEStop
	        OR #iqUDT_EquipmentControl.Command.ResetData
	    THEN

	        "FC_Statistics"(ix_Reset := #iqUDT_EquipmentControl.Command.ResetData,
	                        ix_Activate := #ix_RemotePanelEStop,
	                        ix_RTrigActivate := #sR_Trig_RemotePanelEStop.Q,
	                        iqUDT_Statistics := #iqUDT_Statistics.RemotePanel_EStop);

	    END_IF;


	    //System in error
	    IF #iqUDT_EquipmentControl.Report.Error
	        OR #iqUDT_EquipmentControl.Command.ResetData
	    THEN

	        "FC_Statistics"(ix_Reset := #iqUDT_EquipmentControl.Command.ResetData,
	                        ix_Activate := #iqUDT_EquipmentControl.Report.Error,
	                        ix_RTrigActivate := #sR_TRIG_Error.Q,
	                        iqUDT_Statistics := #iqUDT_Statistics.Error);

	    END_IF;



	    //Number of times start (UPS EMA addition)
	    IF #sR_TRIG_AutomaticOn.Q
	    THEN
	        #iqUDT_Statistics.StartNumberOfTimes += 1;
	    ELSIF #iqUDT_EquipmentControl.Command.ResetData
	    THEN
	        #iqUDT_Statistics.StartNumberOfTimes := 0;
	    END_IF;

	    //Number of times Reset (UPS EMA addition)
	    IF #sF_TRIG_Error.Q
	    THEN
	        #iqUDT_Statistics.ResetNumberOfTimes += 1;
	    ELSIF #iqUDT_EquipmentControl.Command.ResetData
	    THEN
	        #iqUDT_Statistics.ResetNumberOfTimes := 0;
	    END_IF;

	    //Number of times Data Reset (UPS EMA addition)
	    IF #sR_TRIG_DataReset.Q
	    THEN
	        #iqUDT_Statistics.DataResetNumberOfTimes += 1;
	    ELSIF #iqUDT_EquipmentControl.Command.ResetData
	    THEN
	        #iqUDT_Statistics.DataResetNumberOfTimes := 0;
	    END_IF;
	END_REGION

END_FUNCTION_BLOCK

FUNCTION_BLOCK "FB_TCPIPReceive"
TITLE = FB_TCPIPReceive
{ S7_Optimized_Access := 'TRUE' }
AUTHOR : MHSE
FAMILY : Communication
VERSION : 3.0
// ATTRIBUTES
// AUTO_NUMBER = True
// BLOCK_NUMBER = 30
// END_ATTRIBUTES
//Function block to receive data from TCPIP.
// END_ATTRIBUTES
//Function block to receive data from TCPIP.
   VAR_INPUT
      iUDT_Connection { ExternalAccessible := 'False'; ExternalVisible := 'False'; ExternalWritable := 'False'} : "UDT_Connection";   // Connection parameters
      ix_EnableReceive { ExternalAccessible := 'False'; ExternalVisible := 'False'; ExternalWritable := 'False'} : Bool;   // Enable receive
   END_VAR

   VAR_OUTPUT
      qx_Error { ExternalAccessible := 'False'; ExternalVisible := 'False'; ExternalWritable := 'False'} : Bool;   // Collective error output
      qx_Warning { ExternalAccessible := 'False'; ExternalVisible := 'False'; ExternalWritable := 'False'} : Bool;   // Collective warning output
   END_VAR

   VAR_IN_OUT
      iqUDT_FifoHeader : "UDT_FifoHeader";   // Fifo header
      iqUDT_Statistics : "UDT_TCPIPReceiveStatistics";   // Statistic structure
      iqa_FifoData : Array[*] of "UDT_Message";   // Fifo data
   END_VAR

   VAR
      sFB_TRCV {InstructionName := 'TRCV'; LibVersion := '4.0'; ExternalAccessible := 'False'; ExternalVisible := 'False'; ExternalWritable := 'False'; S7_SetPoint := 'False'} : TRCV;   // Siemens "TRCV" block - to receive the data from TCPIP socket
      sa_TRCV { ExternalAccessible := 'False'; ExternalVisible := 'False'; ExternalWritable := 'False'} : Struct   // TRCV block interface structure
         Enable { ExternalAccessible := 'False'; ExternalVisible := 'False'; ExternalWritable := 'False'} : Bool;   //    TRCV - Enable
         NDR { ExternalAccessible := 'False'; ExternalVisible := 'False'; ExternalWritable := 'False'} : Bool;   //    TRCV - New data available
         Busy { ExternalAccessible := 'False'; ExternalVisible := 'False'; ExternalWritable := 'False'} : Bool;   //    TRCV - Busy
         Error { ExternalAccessible := 'False'; ExternalVisible := 'False'; ExternalWritable := 'False'} : Bool;   //    TRCV - Error
         Status { ExternalAccessible := 'False'; ExternalVisible := 'False'; ExternalWritable := 'False'} : Word;   //    TRCV - Status
         RcvLen { ExternalAccessible := 'False'; ExternalVisible := 'False'; ExternalWritable := 'False'} : UDInt;   //    TRCV - Received length
         Data { ExternalAccessible := 'False'; ExternalVisible := 'False'; ExternalWritable := 'False'} : Array[0..999] of Char;   //    TRCV - Data
      END_STRUCT;
      sUDT_MsgArray { ExternalAccessible := 'False'; ExternalVisible := 'False'; ExternalWritable := 'False'; S7_SetPoint := 'False'} : "UDT_Message";   // Message character array
      sUDT_MsgPartArray { ExternalAccessible := 'False'; ExternalVisible := 'False'; ExternalWritable := 'False'; S7_SetPoint := 'False'} : "UDT_Message";   // Part of the message character array
      sa_Status { ExternalAccessible := 'False'; ExternalVisible := 'False'; ExternalWritable := 'False'} : Struct   // Status structure
         ErrorCode { ExternalAccessible := 'False'; ExternalVisible := 'False'; ExternalWritable := 'False'} : Struct   // Error code structure
            TRCV { ExternalAccessible := 'False'; ExternalVisible := 'False'; ExternalWritable := 'False'} : Word;   // Siemens TRCV error code - Check documentation
         END_STRUCT;
         FIFORcvStatus { ExternalAccessible := 'False'; ExternalVisible := 'False'; ExternalWritable := 'False'} : "UDT_FifoStatus";   // Receive FIFO status structure
         FIFORcvError { ExternalAccessible := 'False'; ExternalVisible := 'False'; ExternalWritable := 'False'; S7_SetPoint := 'True'} : Bool;   // Receive FIFO error
         FIFORcvWarning { ExternalAccessible := 'False'; ExternalVisible := 'False'; ExternalWritable := 'False'; S7_SetPoint := 'True'} : Bool;   // Receive  FIFO warning
         ReceiveError { ExternalAccessible := 'False'; ExternalVisible := 'False'; ExternalWritable := 'False'} : Bool;   // TRCV block operation error - Check TRCVStatus
      END_STRUCT;
      sdi_RcvMsgCounter { ExternalAccessible := 'False'; ExternalVisible := 'False'; ExternalWritable := 'False'} : DInt;   // Total received messages counter
      si_RcvMsgOffset { ExternalAccessible := 'False'; ExternalVisible := 'False'; ExternalWritable := 'False'} : Int;   // Received message offset
      si_RcvMsgLen { ExternalAccessible := 'False'; ExternalVisible := 'False'; ExternalWritable := 'False'} : Int;   // Received message length
      si_NrOfRcvMsg { ExternalAccessible := 'False'; ExternalVisible := 'False'; ExternalWritable := 'False'} : Int;   // Number of received messages in one frame
      si_RcvMsgPartLen { ExternalAccessible := 'False'; ExternalVisible := 'False'; ExternalWritable := 'False'} : Int;   // Length of the part of received message
      si_LoopCounter { ExternalAccessible := 'False'; ExternalVisible := 'False'; ExternalWritable := 'False'} : Int;   // Loop counter
      si_MaxMsgLen { ExternalAccessible := 'False'; ExternalVisible := 'False'; ExternalWritable := 'False'} : Int;   // Maximum message length
      sx_RcvMsgPart { ExternalAccessible := 'False'; ExternalVisible := 'False'; ExternalWritable := 'False'} : Bool;   // Received part of the message
      sx_InvalidTermination { ExternalAccessible := 'False'; ExternalVisible := 'False'; ExternalWritable := 'False'} : Bool;   // Termination sign missing
   END_VAR

   VAR CONSTANT
      cc_CRLF_R : Char := '$R';   // First termination sign
      cc_CRLF_L : Char := '$L';   // Last termination sign
      cc_NULL : Char := '$00';   // NULL sign
   END_VAR


BEGIN
	(*
	----------------------------------------------------------------------------------------

	Version history:
	Date        | Version   | Author        | Remark
	----------------------------------------------------------------------------------------
	24/05/2019  | 0.1       | L.Klar        | first release MHS TIA 15.1
	17/06/2019  | 0.3       | A.Nowak       | Replace 2nd level subregions with comments (5.3)
	24/07/2019  | 2.0       | L.Klar        | 2.0 MHS library release TIA 15.1
	22/08/2019  | 2.1       | K.Pokorski    | Comments adjusted
	12/09/2019  | 2.2       | A.Nowak       | Delete buffer size variable
	20/09/2019  | 2.3       | J.Krawczuk    | Replacing UDT_HeartbeatStatus structure to internal structure
	01/10/2019  | 2.4       | A.Nowak       | Implementation of the new FIFO block
	12/11/2019  | 3.0       | P.Majka       | 3.0 MHS library release TIA 15.1
	23/03/2021  | 3.1       | L.Klar        | Static variables data types changed form uint to int
	14/08/2021  | 3.2       | S. Deulkar    | In region 5.3, conveted variable to ULINT because it was giving warning
	21/02/2023  | 4.0       | F.Baten       | 4.0 Release TIA 17.5
	*)

	REGION 1 – Update FIFO header status bits

	    // Mode 'S' - FIFO register status update
	    "FC_Fifo"(ic_Mode := 'S',
	              qUDT_Status => #sa_Status.FIFORcvStatus,
	              qx_Error => #sa_Status.FIFORcvError,
	              qx_Warning => #sa_Status.FIFORcvWarning,
	              iqv_Data := #sUDT_MsgArray,
	              iqUDT_FifoHeader := #iqUDT_FifoHeader,
	              iqv_DataBuffer := #iqa_FifoData);


	END_REGION

	REGION 2 – Maximum number of message arrays elements

	    #si_MaxMsgLen := "FC_GetNrOfArrayEl"(iv_Array := #sUDT_MsgArray.Character);

	END_REGION

	REGION 3 – Receive enable

	    // Allow receiving if the connection is established and there are no fifo errors
	    #sa_TRCV.Enable :=
	    #ix_EnableReceive
	    AND NOT #sa_Status.FIFORcvError;

	END_REGION

	REGION 4 – Receive data

	    // Data received in an ADHOC mode - data available immediately
	    #sFB_TRCV(EN_R := #sa_TRCV.Enable,
	              ID := #iUDT_Connection.ID,
	              LEN := 0,
	              ADHOC := TRUE,
	              NDR => #sa_TRCV.NDR,
	              BUSY => #sa_TRCV.Busy,
	              ERROR => #sa_TRCV.Error,
	              STATUS => #sa_TRCV.Status,
	              RCVD_LEN => #sa_TRCV.RcvLen,
	              DATA := #sa_TRCV.Data);

	END_REGION

	IF #sa_TRCV.RcvLen > 1000 THEN
	    #sa_TRCV.RcvLen := 1000;
	END_IF;

	REGION 5 – Received data handling

	    // Receiving data was successful
	    IF (#sa_TRCV.NDR                    // New data received without error
	        AND NOT #sa_TRCV.Busy           // Job not yet started or already completed
	        AND NOT #sa_TRCV.Error          // No errors during receiving messages
	        AND #sa_TRCV.RcvLen > 0)        // Length greater than zero
	    THEN

	        REGION 5.1 – Initialization

	            #si_RcvMsgLen := 0;
	            #si_RcvMsgOffset := 0;
	            #si_NrOfRcvMsg := 0;

	        END_REGION

	        REGION 5.2 – Received part of the message

	            // Move part of the messages to a buffer if available
	            IF (#sx_RcvMsgPart)                             // Message part available
	            THEN

	                #sUDT_MsgArray := #sUDT_MsgPartArray;
	                #sx_RcvMsgPart := FALSE;

	            END_IF;

	        END_REGION

	        REGION 5.3 – Message handling

	            FOR #si_LoopCounter := 0 TO UDINT_TO_INT(#sa_TRCV.RcvLen) - 1 DO

	                // Message length validation
	                IF (#si_RcvMsgLen + #si_RcvMsgPartLen < #si_MaxMsgLen)
	                THEN

	                    // Termination sign found
	                    IF (#sa_TRCV.Data[#si_LoopCounter] = #cc_CRLF_L)
	                    THEN

	                        // Move received message to the message array
	                        MOVE_BLK(IN := #sa_TRCV.Data[#si_RcvMsgOffset],
	                                 COUNT := INT_TO_ULINT(#si_RcvMsgLen),
	                                 OUT => #sUDT_MsgArray.Character[#si_RcvMsgPartLen]);

	                        // Clear NOT used message array characters
	                        FILL_BLK(IN := #cc_NULL,
	                                 COUNT := INT_TO_ULINT(#si_MaxMsgLen - #si_RcvMsgLen + #si_RcvMsgPartLen),
	                                 OUT => #sUDT_MsgArray.Character[#si_RcvMsgLen + #si_RcvMsgPartLen]);

	                        // Check and clear termination sign
	                        IF (#si_RcvMsgLen + #si_RcvMsgPartLen - 1) >= 0 AND (#si_RcvMsgLen + #si_RcvMsgPartLen - 1) < #si_MaxMsgLen THEN
	                            IF (#sUDT_MsgArray.Character[#si_RcvMsgLen + #si_RcvMsgPartLen - 1] = #cc_CRLF_R)        // Character is a termination sign
	                            THEN

	                                #sUDT_MsgArray.Character[#si_RcvMsgLen + #si_RcvMsgPartLen - 1] := #cc_NULL;

	                                // Termination sign invalid - error generated, statistics increased
	                            ELSE

	                                #sx_InvalidTermination := TRUE;
	                                #iqUDT_Statistics.InvalidMsg += 1;

	                            END_IF;
	                        ELSE
	                            #iqUDT_Statistics.InvalidMsg += 1;
	                        END_IF;


	                        // Move message into the FIFO data block
	                        IF (NOT #sx_InvalidTermination)                                         // No termination sign error
	                        THEN

	                            // Mode 'W' - Write FIFO record
	                            "FC_Fifo"(ic_Mode := 'W',
	                                      qUDT_Status => #sa_Status.FIFORcvStatus,
	                                      qx_Error => #sa_Status.FIFORcvError,
	                                      qx_Warning => #sa_Status.FIFORcvWarning,
	                                      iqv_Data := #sUDT_MsgArray,
	                                      iqUDT_FifoHeader := #iqUDT_FifoHeader,
	                                      iqv_DataBuffer := #iqa_FifoData);


	                        END_IF;

	                        #sx_InvalidTermination := FALSE;                                    // Reset the invalid termination bit

	                        // Update lengths and counters
	                        #si_RcvMsgPartLen := 0;
	                        #si_RcvMsgOffset += #si_RcvMsgLen + 1;
	                        #si_RcvMsgLen := 0;
	                        #si_NrOfRcvMsg += 1;
	                        #sdi_RcvMsgCounter += 1;

	                        // Termination sign not found
	                    ELSE

	                        #si_RcvMsgLen := #si_RcvMsgLen + 1;                               // Increment received message length

	                    END_IF;

	                    // Message length invalid - reset message length and increase statistics
	                ELSE

	                    #si_RcvMsgLen := 0;
	                    #iqUDT_Statistics.InvalidMsg += 1;

	                END_IF;

	            END_FOR;

	        END_REGION

	        REGION 5.4 – Part of the message preparation


	            // Move part of the message to buffer when last received sign is not a termination signs
	            IF (#sa_TRCV.Data[UDINT_TO_INT(#sa_TRCV.RcvLen - 1)] <> #cc_CRLF_L            // Last received sign is not a termination sing
	                AND #si_RcvMsgLen < #si_MaxMsgLen)                         // Message length valid
	            THEN

	                // Fill not used message char array elements with '$00'
	                FILL_BLK(IN := '$00',
	                         COUNT := INT_TO_ULINT(#si_MaxMsgLen) -
	                         INT_TO_ULINT(#si_RcvMsgLen),
	                         OUT => #sUDT_MsgPartArray.Character[#si_RcvMsgLen]);

	                // Move part of the message to a buffer
	                MOVE_BLK(IN := #sa_TRCV.Data[#si_RcvMsgOffset],
	                         COUNT := INT_TO_ULINT(#si_RcvMsgLen),
	                         OUT => #sUDT_MsgPartArray.Character[0]);

	                // Set the part of the message received bit and move length of the received message into the length of the part of the message variable
	                #sx_RcvMsgPart := TRUE;
	                #si_RcvMsgPartLen := #si_RcvMsgLen;

	            END_IF;

	        END_REGION

	    END_IF;

	END_REGION

	REGION 6 – Status

	    REGION 6.1 - Block status

	        // Receive error
	        #sa_Status.ReceiveError := #sa_TRCV.Error;

	        // Parametrization collective error output
	        #qx_Error :=
	        #sa_Status.FIFORcvError                          // FIFO error
	        OR #sa_Status.ReceiveError;                      // Receive error

	        // Parametrization collective warning output
	        #qx_Warning := #sa_Status.FIFORcvWarning;        // FIFO warning

	    END_REGION

	    REGION 6.2 - Error code preparation

	        IF (#sa_TRCV.#Status > 16#8000
	            OR #sa_TRCV.#Status = 16#0)
	        THEN

	            #sa_Status.ErrorCode.TRCV := #sa_TRCV.#Status;

	        END_IF;

	    END_REGION

	END_REGION
END_FUNCTION_BLOCK

FUNCTION_BLOCK "FB_TCPIPSend"
TITLE = FB_TCPIPSend
{ S7_Optimized_Access := 'TRUE' }
AUTHOR : MHSE
FAMILY : Communication
VERSION : 3.0
// ATTRIBUTES
// AUTO_NUMBER = True
// BLOCK_NUMBER = 31
// END_ATTRIBUTES
//Function block to send data from TCPIP.
   VAR_INPUT
      iUDT_Connection { ExternalAccessible := 'False'; ExternalVisible := 'False'; ExternalWritable := 'False'} : "UDT_Connection";   // Connection parameters
      ix_EnableSend { ExternalAccessible := 'False'; ExternalVisible := 'False'; ExternalWritable := 'False'} : Bool;   // Enable send
   END_VAR

   VAR_OUTPUT
      qx_Error { ExternalAccessible := 'False'; ExternalVisible := 'False'; ExternalWritable := 'False'} : Bool;   // Collective error output
      qx_Warning { ExternalAccessible := 'False'; ExternalVisible := 'False'; ExternalWritable := 'False'} : Bool;   // Collective warning output
   END_VAR

   VAR_IN_OUT
      iqUDT_FifoLowHeader : "UDT_FifoHeader";   // Low priority FIFO header
      iqs_FifoLowData : Array[*] of "UDT_Message";   // Low priority FIFO data
      iqUDT_FifoMedHeader : "UDT_FifoHeader";   // Medium priority FIFO header
      iqs_FifoMedData : Array[*] of "UDT_Message";   // Medium priority FIFO data
      iqUDT_FifoHighHeader : "UDT_FifoHeader";   // High priority FIFO header
      iqs_FifoHighData : Array[*] of "UDT_Message";   // High priority FIFO data
   END_VAR

   VAR
      sFB_TSEND {InstructionName := 'TSEND'; LibVersion := '4.0'; ExternalAccessible := 'False'; ExternalVisible := 'False'; ExternalWritable := 'False'; S7_SetPoint := 'False'} : TSEND;   // Siemens "TSEND" block - to send the data over TCPIP socket
      sUDT_MsgArray { ExternalAccessible := 'False'; ExternalVisible := 'False'; ExternalWritable := 'False'; S7_SetPoint := 'False'} : "UDT_Message";   // Message character array
      sa_TSEND { ExternalAccessible := 'False'; ExternalVisible := 'False'; ExternalWritable := 'False'} : Struct   // TSEND block structure
         Status { ExternalAccessible := 'False'; ExternalVisible := 'False'; ExternalWritable := 'False'} : Word;   // TSEND - Status
         Request { ExternalAccessible := 'False'; ExternalVisible := 'False'; ExternalWritable := 'False'} : Bool;   // TSEND - Request
         Busy { ExternalAccessible := 'False'; ExternalVisible := 'False'; ExternalWritable := 'False'} : Bool;   // TSEND - Busy
         Done { ExternalAccessible := 'False'; ExternalVisible := 'False'; ExternalWritable := 'False'} : Bool;   // TSEND - Done
         Error { ExternalAccessible := 'False'; ExternalVisible := 'False'; ExternalWritable := 'False'} : Bool;   //  TSEND - Error
      END_STRUCT;
      sa_Status { ExternalAccessible := 'False'; ExternalVisible := 'False'; ExternalWritable := 'False'} : Struct   // Status structure
         FIFOLowPrioStatus { ExternalAccessible := 'False'; ExternalVisible := 'False'; ExternalWritable := 'False'} : "UDT_FifoStatus";
         FIFOMedPrioStatus { ExternalAccessible := 'False'; ExternalVisible := 'False'; ExternalWritable := 'False'} : "UDT_FifoStatus";
         FIFOHighPrioStatus { ExternalAccessible := 'False'; ExternalVisible := 'False'; ExternalWritable := 'False'} : "UDT_FifoStatus";
         FIFOLowPrioError { ExternalAccessible := 'False'; ExternalVisible := 'False'; ExternalWritable := 'False'} : Bool;   // FIFO low priority error
         FIFOLowPrioWarning { ExternalAccessible := 'False'; ExternalVisible := 'False'; ExternalWritable := 'False'} : Bool;   // FIFO low priority warning
         FIFOMedPrioError { ExternalAccessible := 'False'; ExternalVisible := 'False'; ExternalWritable := 'False'} : Bool;   // FIFO medium priority error
         FIFOMedPrioWarning { ExternalAccessible := 'False'; ExternalVisible := 'False'; ExternalWritable := 'False'} : Bool;   // FIFO medium priority warning
         FIFOHighPrioError { ExternalAccessible := 'False'; ExternalVisible := 'False'; ExternalWritable := 'False'} : Bool;   // FIFO high priority error
         FIFOHighPrioWarning { ExternalAccessible := 'False'; ExternalVisible := 'False'; ExternalWritable := 'False'} : Bool;   // FIFO high priority warning
         SendError { ExternalAccessible := 'False'; ExternalVisible := 'False'; ExternalWritable := 'False'} : Bool;   // Send operation error
      END_STRUCT;
      si_MaxMsgLen { ExternalAccessible := 'False'; ExternalVisible := 'False'; ExternalWritable := 'False'} : Int;   // Maximum message length
      si_MsgLen { ExternalAccessible := 'False'; ExternalVisible := 'False'; ExternalWritable := 'False'} : Int;   // Message length
      sx_MsgReady { ExternalAccessible := 'False'; ExternalVisible := 'False'; ExternalWritable := 'False'} : Bool;   // Message is ready to send
      sx_MsgRead { ExternalAccessible := 'False'; ExternalVisible := 'False'; ExternalWritable := 'False'} : Bool;   // Message has been read
      sx_MsgReadReq { ExternalAccessible := 'False'; ExternalVisible := 'False'; ExternalWritable := 'False'} : Bool;   // Request to read message
      sx_FIFOError { ExternalAccessible := 'False'; ExternalVisible := 'False'; ExternalWritable := 'False'} : Bool;   // Summary FIFO error
   END_VAR

   VAR CONSTANT
      cc_NULL : Char := '$00';   // NULL sign
   END_VAR


BEGIN
	(*
	----------------------------------------------------------------------------------------

	Version history:
	Date        | Version   | Author        | Remark
	----------------------------------------------------------------------------------------
	24/05/2019  | 0.1       | L.Klar        | first release MHS TIA 15.1
	13/06/2019  | 0.2       | A.Nowak       | Replacement of instruction if for direct write into variable - Region 7
	25/06/2019  | 0.5       | L.Klar        | Comments corrected
	18/07/2019  | 0.6       | L.Klar        | Status handling changed
	24/07/2019  | 2.0       | L.Klar        | 2.0 MHS library release TIA 15.1
	22/08/2019  | 2.1       | K.Pokorski    | Comments adjusted
	20/09/2019  | 2.2       | K.Pokorski    | "UDT_Status" deleted
	26/09/2019  | 2.3       | A.Nowak       | Delete NoDataTOSend and TSEND status code from status structure. Delete region 7.
	02/10/2019  | 2.4       | A.Nowak       | Implementation of the new FIFO block
	12/11/2019  | 3.0       | P.Majka       | 3.0 MHS library release TIA 15.1
	21/02/2023  | 4.0       | F.Baten       | 4.0 Release TIA 17.5
	*)

	REGION 1 – Update FIFO header status bits

	    // Mode 'S' - High priority FIFO register status update
	    "FC_Fifo"(ic_Mode := 'S',
	              qUDT_Status => #sa_Status.FIFOHighPrioStatus,
	              qx_Error => #sa_Status.FIFOHighPrioError,
	              qx_Warning => #sa_Status.FIFOHighPrioWarning,
	              iqv_Data := #sUDT_MsgArray,
	              iqUDT_FifoHeader := #iqUDT_FifoHighHeader,
	              iqv_DataBuffer := #iqs_FifoHighData);


	    // Mode 'S' - Medium priority FIFO register status update
	    "FC_Fifo"(ic_Mode := 'S',
	              qUDT_Status => #sa_Status.FIFOMedPrioStatus,
	              qx_Error => #sa_Status.FIFOMedPrioError,
	              qx_Warning => #sa_Status.FIFOMedPrioWarning,
	              iqv_Data := #sUDT_MsgArray,
	              iqUDT_FifoHeader := #iqUDT_FifoMedHeader,
	              iqv_DataBuffer := #iqs_FifoMedData);

	    // Mode 'S' - Low priority FIFO register status update
	    "FC_Fifo"(ic_Mode := 'S',
	              qUDT_Status => #sa_Status.FIFOLowPrioStatus,
	              qx_Error => #sa_Status.FIFOLowPrioError,
	              qx_Warning => #sa_Status.FIFOLowPrioWarning,
	              iqv_Data := #sUDT_MsgArray,
	              iqUDT_FifoHeader := #iqUDT_FifoLowHeader,
	              iqv_DataBuffer := #iqs_FifoLowData);

	END_REGION

	REGION 2 – FIFO header summary error

	    #sx_FIFOError :=
	    #sa_Status.FIFOHighPrioError         // High priority FIFO error
	    OR #sa_Status.FIFOMedPrioError       // Medium priority FIFO error
	    OR #sa_Status.FIFOLowPrioError;      // Low priority FIFO error

	END_REGION

	REGION 3 – FIFO Read request

	    #sx_MsgReadReq :=
	    #ix_EnableSend                      // Connection is established
	    AND NOT #sx_FIFOError               // No FIFO errors
	    AND NOT #sa_TSEND.Error             // No TSEND errors
	    AND #sa_TSEND.Status = 16#7000;     // TSEND block status equal to 16#7000 - no job

	END_REGION

	REGION 4 – Read the message from high priority FIFO data buffer

	    IF (#sx_MsgReadReq                                                          // Read request
	        AND NOT #iqUDT_FifoHighHeader.Status.Empty                             // High priority FIFO data buffer is not empty
	        AND NOT #sx_MsgRead)                                                    // Message isn't read
	    THEN

	        // Mode 'R' - Read high priority FIFO record
	        "FC_Fifo"(ic_Mode := 'R',
	                  qUDT_Status => #sa_Status.FIFOHighPrioStatus,
	                  qx_Error => #sa_Status.FIFOHighPrioError,
	                  qx_Warning => #sa_Status.FIFOHighPrioWarning,
	                  iqv_Data := #sUDT_MsgArray,
	                  iqUDT_FifoHeader := #iqUDT_FifoHighHeader,
	                  iqv_DataBuffer := #iqs_FifoHighData);

	        #sx_MsgRead := TRUE;                                                        // Message read bit

	    END_IF;

	END_REGION

	REGION 5 – Read the message from medium priority FIFO data buffer

	    IF (#sx_MsgReadReq                                                              // Read request,
	        AND #iqUDT_FifoHighHeader.Status.Empty                                     // High priority FIFO data buffer empty
	        AND NOT #iqUDT_FifoMedHeader.Status.Empty                                  // Medium priority FIFO data buffer not empty
	        AND NOT #sx_MsgRead)                                                        // Message not read
	    THEN

	        // Mode 'R' - Read medium priority FIFO record
	        "FC_Fifo"(ic_Mode := 'R',
	                  qUDT_Status => #sa_Status.FIFOMedPrioStatus,
	                  qx_Error => #sa_Status.FIFOMedPrioError,
	                  qx_Warning => #sa_Status.FIFOMedPrioWarning,
	                  iqv_Data := #sUDT_MsgArray,
	                  iqUDT_FifoHeader := #iqUDT_FifoMedHeader,
	                  iqv_DataBuffer := #iqs_FifoMedData);

	        #sx_MsgRead := TRUE;                                                        // Message read bit

	    END_IF;

	END_REGION

	REGION 6 – Read the message from low priority FIFO data buffer

	    IF (#sx_MsgReadReq                                                          // Read request
	        AND #iqUDT_FifoHighHeader.Status.Empty                                 // High priority FIFO data buffer empty
	        AND #iqUDT_FifoMedHeader.Status.Empty                                  // Medium priority FIFO data buffer empty
	        AND NOT #iqUDT_FifoLowHeader.Status.Empty                              // Low priority FIFO data buffer not empty
	        AND NOT #sx_MsgRead)                                                    // Message not read
	    THEN

	        #sx_MsgRead := TRUE;                                                    // Message read bit

	        // Mode 'R' - Read low priority FIFO record
	        "FC_Fifo"(ic_Mode := 'R',
	                  qUDT_Status => #sa_Status.FIFOLowPrioStatus,
	                  qx_Error => #sa_Status.FIFOLowPrioError,
	                  qx_Warning => #sa_Status.FIFOLowPrioWarning,
	                  iqv_Data := #sUDT_MsgArray,
	                  iqUDT_FifoHeader := #iqUDT_FifoLowHeader,
	                  iqv_DataBuffer := #iqs_FifoLowData);

	    END_IF;

	END_REGION

	REGION 7 – Maximum number of message array elements

	    #si_MaxMsgLen := "FC_GetNrOfArrayEl"(iv_Array := #sUDT_MsgArray.Character);

	END_REGION

	REGION 8 – Message length

	    // Measuring the length of a read message
	    IF (#sx_MsgRead                                                 // The message is read
	        AND NOT #sx_MsgReady)                                       // The message is not ready
	    THEN

	        // Initialize the message length
	        #si_MsgLen := 0;

	        // Message character counting loop
	        WHILE #sUDT_MsgArray.Character[#si_MsgLen] <> #cc_NULL     // Message array character is diffrent then NULL sign
	            AND #si_MsgLen < #si_MaxMsgLen - 1                      // Message length is lower then maximum message length minus 1
	        DO

	            #si_MsgLen += 1;

	        END_WHILE;

	        #sx_MsgReady := TRUE;

	    END_IF;

	END_REGION

	REGION 9 – Send request

	    IF (#sx_MsgRead                     // The message is read
	        AND #sx_MsgReady)               // The message is ready

	    THEN

	        #sa_TSEND.Request := TRUE;

	    END_IF;

	END_REGION

	REGION 10 – Send data

	    #sFB_TSEND(REQ := #sa_TSEND.Request,
	               ID := #iUDT_Connection.ID,
	               LEN := INT_TO_UDINT(#si_MsgLen),
	               DONE => #sa_TSEND.Done,
	               BUSY => #sa_TSEND.Busy,
	               ERROR => #sa_TSEND.Error,
	               STATUS => #sa_TSEND.Status,
	               DATA := #sUDT_MsgArray);

	    // Reset send request, message read and ready bits
	    IF (#sa_TSEND.Request                                       // Send request
	        AND NOT #sa_TSEND.Busy                                  // TSEND block not busy
	        AND (#sa_TSEND.Done                                     // Send operation done
	        OR #sa_TSEND.Status = 16#7000))                     // Communication is not established
	    THEN

	        #sa_TSEND.Request := FALSE;
	        #sx_MsgRead := FALSE;
	        #sx_MsgReady := FALSE;

	    END_IF;

	    // Reset send error and TSEND status after correctly sent message
	    IF (#sa_TSEND.Done)                                                 // Send operation done
	    THEN

	        #sa_Status.SendError := FALSE;

	    END_IF;

	    // Set send error and TSEND status if error occured
	    IF (#sa_TSEND.Error)                                                // TSEND error
	    THEN

	        #sa_Status.SendError := TRUE;

	    END_IF;

	END_REGION

	REGION 11 – Status

	    // Parametrization collective error output
	    #qx_Error :=
	    #sx_FIFOError                           // FIFO errors and
	    OR #sa_Status.SendError;                // TSEND block operation error

	    // Parametrization collective warning output
	    #qx_Warning :=
	    #sa_Status.FIFOHighPrioWarning          // High priority FIFO warning bit
	    OR #sa_Status.FIFOMedPrioWarning        // Medium priority FIFO warning bit
	    OR #sa_Status.FIFOLowPrioWarning;       // Low priority FIFO warning bit

	END_REGION
END_FUNCTION_BLOCK

FUNCTION_BLOCK "FB_Tracking"
TITLE = FB_Tracking
{ S7_Optimized_Access := 'TRUE' }
AUTHOR : MHSE
FAMILY : GeneralSystemFunctions
VERSION : 3.0
// ATTRIBUTES
// AUTO_NUMBER = True
// BLOCK_NUMBER = 33
// END_ATTRIBUTES
//Function block to shift data in the tracking array.
   VAR_INPUT
      iUDT_ConveyorCommonConfiguration { ExternalAccessible := 'False'; ExternalVisible := 'False'; ExternalWritable := 'False'} : "UDT_ConveyorCommonConfiguration";   // Conveyor common configuration
   END_VAR

   VAR_IN_OUT
      iqa_TrackingData : Array[*] of Int;   // Tracking array
      iqUDT_ConveyorInterface : "UDT_ConveyorInterface";   // Conveyor interface
      iqUDT_HandshakeUp : "UDT_ConveyorHandshake";   // Upstream conveyor handshake
      iqUDT_Handshake : "UDT_ConveyorHandshake";   // Conveyor handshake
   END_VAR

   VAR
      si_TrackingArrayLen { ExternalAccessible := 'False'; ExternalVisible := 'False'; ExternalWritable := 'False'} : Int;   // Tracking array length
      si_TrackingArrayLowBound { ExternalAccessible := 'False'; ExternalVisible := 'False'; ExternalWritable := 'False'} : Int;   // Tracking array lower bound
      sdi_TotalConvLength { ExternalAccessible := 'False'; ExternalVisible := 'False'; ExternalWritable := 'False'} : DInt;   // Number of tracking entries is equal to the conveyor length in cm
      si_Displacement { ExternalAccessible := 'False'; ExternalVisible := 'False'; ExternalWritable := 'False'} : Int;   // Displacement
      si_ShiftDestination { ExternalAccessible := 'False'; ExternalVisible := 'False'; ExternalWritable := 'False'} : Int;   // Pointer to the entry to start writing the tracking data
      si_ShiftOffset { ExternalAccessible := 'False'; ExternalVisible := 'False'; ExternalWritable := 'False'} : Int;   // Number of entries to be shifted and its direction
      sdi_GINInsertPosition { ExternalAccessible := 'False'; ExternalVisible := 'False'; ExternalWritable := 'False'} : DInt;   // Position where GIN form upstream conveyor will be inserted
      sdi_GINExtractPosition { ExternalAccessible := 'False'; ExternalVisible := 'False'; ExternalWritable := 'False'} : DInt;   // Position from which GIN will be moved to the downstream conveyor
      sx_InvalidTrackArraySize { ExternalAccessible := 'False'; ExternalVisible := 'False'; ExternalWritable := 'False'} : Bool;   // Invalid tracking array size
   END_VAR


BEGIN
	(*
	----------------------------------------------------------------------------------------
	|                                                                                      |
	|  Copyright  2019             MHS                                                     |
	|  All Rights Reserved         Larenweg 90                                             |
	|                              5234 KC 's-Hertogenbosch,                               |
	|                              Netherlands                                             |
	|                                                                                      |
	----------------------------------------------------------------------------------------

	Version history:
	Date        | Version   | Author       | Remark
	----------------------------------------------------------------------------------------
	24/05/2019  | 0.1       | L. Klar      | first release MHS TIA 15.1
	14/06/2019  | 0.2       | A.Nowak      | Replacement of instruction if for direct write into variable - Region 3
	19/07/2019  | 0.5       | L.Klar       | Status handling changed
	24/07/2019  | 2.0       | L.Klar       | 2.0 MHS library release TIA 15.1
	23/08/2019  | 2.1       | L.Klar       | "UDT_ConveyorConfiguration" changed to "UDT_ConveyorCommonConfiguration", internal tracking error set instead of coil assigment.
	10/09/2019  | 2.2       | L.Klar       | Comments changed, block optimized
	21/10/2019  | 2.3       | L.Klar       | Configuration UDT chanaged to input
	12/11/2019  | 3.0       | P.Majka      | 3.0 MHS library release TIA 15.1
	20/12/2019  | 3.1       | S. Deulkar   | Used configureation error bit to report to conveyor block
	15/01/2020  | 3.2       | L.Klar       | Block adjusted to allow to transfer negative GIN numbers
	*)

	REGION 1 – Get the required number of entries

	    // Number of entries is a conveyor length in cm
	    #sdi_TotalConvLength := (#iUDT_ConveyorCommonConfiguration.Length + #iUDT_ConveyorCommonConfiguration.LengthCorrection) / 10;

	END_REGION

	REGION 2 – Number of tracking records validation

	    // Tracking array dimensions
	    #si_TrackingArrayLen := "FC_GetNrOfArrayEl"(#iqa_TrackingData);
	    #si_TrackingArrayLowBound := DINT_TO_INT(LOWER_BOUND(ARR := #iqa_TrackingData, DIM := 1));

	    // Check if the number of entries is exceeding the tracking array size
	    #sx_InvalidTrackArraySize := #si_TrackingArrayLen < #sdi_TotalConvLength + 2
	    OR #si_TrackingArrayLowBound <> 0;

	END_REGION

	REGION 3 – Read the displacement

	    #si_Displacement := #iqUDT_ConveyorInterface.Displacement;

	END_REGION

	REGION 4 – Prepare tracking array pointers

	    // A conveyor can run in forward and reverse direction
	    // Data will be shifted into tracking entry position 1 for both cases.
	    #si_ShiftDestination := 1;

	    // If the direction is forward (positive displacement), entry 2 is taken as offset (shifts conveyor length from pos 2 in pos 1)
	    IF #si_Displacement > 0
	    THEN

	        #si_ShiftOffset := 2;
	        #sdi_GINInsertPosition := #sdi_TotalConvLength + 1;
	        #sdi_GINExtractPosition := 1;

	        // If the direction is reverse (negative displacement), entry 0 is taken as offset (shifts conveyor length from pos 0 in pos 1)
	    ELSE

	        #si_ShiftOffset := 0;
	        #sdi_GINInsertPosition := 0;
	        #sdi_GINExtractPosition := #sdi_TotalConvLength;

	    END_IF;

	END_REGION

	REGION 5 – Shift data

	    // Data is shifted only if the conveyor is running (positive or negtive displacement)
	    WHILE #si_Displacement <> 0 DO

	        // Conveyor running forward
	        IF (#si_Displacement > 0)
	        THEN

	            // GIN is moved into the tracking array on GIN insert position if the number of positions in upstream conveyor handshake is available
	            // The number of positions to be shifted will be decremented
	            IF (#iqUDT_HandshakeUp.GIN <> 0
	                AND #iqUDT_HandshakeUp.NrOfPosToShift > 0)
	            THEN

	                #iqa_TrackingData[#sdi_GINInsertPosition] := #iqUDT_HandshakeUp.GIN;
	                #iqUDT_HandshakeUp.NrOfPosToShift -= 1;

	            ELSIF (#iqUDT_HandshakeUp.GIN <> 0
	                AND #iqUDT_HandshakeUp.NrOfPosToShift = 0)
	            THEN

	                #iqa_TrackingData[#sdi_GINInsertPosition] := #iqUDT_HandshakeUp.GIN;

	            END_IF;

	            // Clear the downsteam handshake GIN if the number of positions to be shifted is 0
	            IF (#iqUDT_Handshake.GIN <> 0 AND #iqUDT_Handshake.NrOfPosToShift = 0)
	            THEN

	                #iqUDT_Handshake.GIN := 0;

	            END_IF;

	            // GIN is moved into the handshake structure if the data is available at GIN extract position
	            // The number of positions will be incremented
	            IF (#iqa_TrackingData[#sdi_GINExtractPosition] <> 0)
	            THEN

	                IF (#iqUDT_Handshake.GIN = 0)
	                THEN

	                    #iqUDT_Handshake.GIN := #iqa_TrackingData[#sdi_GINExtractPosition];
	                    #iqUDT_Handshake.NrOfPosToShift += 1;

	                ELSIF (#iqUDT_Handshake.GIN = #iqa_TrackingData[#sdi_GINExtractPosition])
	                THEN

	                    #iqUDT_Handshake.NrOfPosToShift += 1;

	                END_IF;

	            END_IF;

	            // Update displacement
	            #si_Displacement -= 1;

	            // Conveyor running backward
	        ELSIF (#si_Displacement < 0)
	        THEN

	            // GIN is moved into the tracking array on GIN insert position if the number of positions in downstream conveyor handshake is available
	            // The number of positions to be shifted will be decremented
	            IF (#iqUDT_Handshake.GIN <> 0
	                AND #iqUDT_Handshake.NrOfPosToShift > 0)
	            THEN

	                #iqa_TrackingData[#sdi_GINInsertPosition] := #iqUDT_Handshake.GIN;
	                #iqUDT_Handshake.NrOfPosToShift -= 1;

	                // In case of displacement greater than 1 and no positions to be shifted the GIN will be written to avoid gaps in data
	                // Writing will be stopped when GIN 0 is detected
	            ELSIF (#iqUDT_Handshake.GIN <> 0
	                AND #iqUDT_Handshake.NrOfPosToShift = 0)
	            THEN

	                #iqa_TrackingData[#sdi_GINInsertPosition] := #iqUDT_Handshake.GIN;

	            END_IF;

	            // Clear the upstream handshake GIN if the number of positions to be shifted is 0
	            IF (#iqUDT_HandshakeUp.GIN <> 0 AND #iqUDT_HandshakeUp.NrOfPosToShift = 0)
	            THEN

	                #iqUDT_HandshakeUp.GIN := 0;

	            END_IF;

	            // GIN is moved into the handshake structure if the data is available at GIN extract position
	            // The number of positions will be incremented
	            IF (#iqa_TrackingData[#sdi_GINExtractPosition] <> 0)
	            THEN

	                IF (#iqUDT_HandshakeUp.GIN = 0)
	                THEN

	                    #iqUDT_HandshakeUp.GIN := #iqa_TrackingData[#sdi_GINExtractPosition];
	                    #iqUDT_HandshakeUp.NrOfPosToShift += 1;

	                    // In case of displacement greater than 1 and no positions to be shifted the GIN will be written to avoid gaps in data
	                    // Writing will be stopped when GIN 0 is detected
	                ELSIF (#iqUDT_HandshakeUp.GIN = #iqa_TrackingData[#sdi_GINExtractPosition])
	                THEN

	                    #iqUDT_HandshakeUp.NrOfPosToShift += 1;

	                END_IF;

	            END_IF;

	            // Update displacement
	            #si_Displacement += 1;

	        END_IF;

	        // Shift the total conveyor length (number of tracking array entries) one cm up or down
	        MOVE_BLK(IN := #iqa_TrackingData[#si_ShiftOffset],
	                 COUNT := DINT_TO_ULINT(#sdi_TotalConvLength),
	                 OUT => #iqa_TrackingData[#si_ShiftDestination]);

	        // Clear the GIN insert position
	        #iqa_TrackingData[#sdi_GINInsertPosition] := 0;

	    END_WHILE;

	END_REGION

	REGION 6 – Internal tracking error

	    // The internal tracking error is set to stop the conveyor
	    // It is reset in the conveyor block
	    IF (#sx_InvalidTrackArraySize)
	    THEN

	        #iqUDT_ConveyorInterface.ConfigurationError := TRUE;

	    END_IF;

	END_REGION
END_FUNCTION_BLOCK

FUNCTION_BLOCK "FB_PECBulkD"
TITLE = FB_PEC
{ S7_Optimized_Access := 'TRUE' }
AUTHOR : MHSE
FAMILY : Conveyor
VERSION : 3.0
// ATTRIBUTES
// AUTO_NUMBER = True
// BLOCK_NUMBER = 21
// END_ATTRIBUTES
   VAR_INPUT
      iUDT_PECConfiguration { ExternalAccessible := 'False'; ExternalVisible := 'False'; ExternalWritable := 'False'} : "UDT_PECDConfiguration";   //   PEC configuration structure
      ix_PEC { ExternalAccessible := 'False'; ExternalVisible := 'False'; ExternalWritable := 'False'} : Bool;   //   Signal of the PEC
      ix_PECDownstream { ExternalAccessible := 'False'; ExternalVisible := 'False'; ExternalWritable := 'False'} : Bool;   //   Downstream PEC signal
      ix_DownstreamRunning { ExternalAccessible := 'False'; ExternalVisible := 'False'; ExternalWritable := 'False'} : Bool;   //  Downstream conveyor is running
   END_VAR

   VAR_OUTPUT
      qUDT_HMIStatus { ExternalAccessible := 'False'; ExternalVisible := 'False'; ExternalWritable := 'False'} : "UDT_PECStatus";   //   Status structure
      qx_PECFiltered { ExternalAccessible := 'False'; ExternalVisible := 'False'; ExternalWritable := 'False'} : Bool;   //   PEC Filtered
   END_VAR

   VAR_IN_OUT
      iqUDT_ConveyorInterface : "UDT_ConveyorInterface";   //   Interface structure
      iqUDT_PECStatistics : "UDT_PECStatistics";   //   Statistics structure
   END_VAR

   VAR
      s_Status { ExternalAccessible := 'False'; ExternalVisible := 'False'; ExternalWritable := 'False'; S7_SetPoint := 'False'} : "UDT_PECStatus";   //   Status structure
      s_StatusOld { ExternalAccessible := 'False'; ExternalVisible := 'False'; ExternalWritable := 'False'; S7_SetPoint := 'False'} : "UDT_PECStatus";   //   Auxiliary status structure
      PEC_OnOffDelay { ExternalAccessible := 'False'; ExternalVisible := 'False'; ExternalWritable := 'False'; S7_SetPoint := 'False'} : "FB_OnOffDelayDistance";   //   Filtering end of section photo eye signal
      R_TRIG_PECJam {InstructionName := 'R_TRIG'; LibVersion := '1.0'; ExternalAccessible := 'False'; ExternalVisible := 'False'; ExternalWritable := 'False'; S7_SetPoint := 'False'} : R_TRIG;   //   Rising edge trigger PEC jam
   END_VAR
   VAR RETAIN
      si_AuxJamDisplacement { ExternalAccessible := 'False'; ExternalVisible := 'False'; ExternalWritable := 'False'} : Int;   //   Auxiliary variable to calculate displacement when PEC is blocked
   END_VAR
   VAR
      sx_Enable { ExternalAccessible := 'False'; ExternalVisible := 'False'; ExternalWritable := 'False'} : Bool;   //   Enable
      sx_PECFiltered { ExternalAccessible := 'False'; ExternalVisible := 'False'; ExternalWritable := 'False'} : Bool;   //   Photo eye filtered
   END_VAR


BEGIN
	(*
	----------------------------------------------------------------------------------------

	Version history:
	Date        | Version   | Author        | Remark
	----------------------------------------------------------------------------------------
	 16/03/2020 | 3.0       | K.Pokorski    | 3.0 MHS library release TIA 15.1
	 20/03/2020 | 3.1       | S.Theocharis  | Changed check to upsteam and jam condition
	 24/03/2020 | 3.2       | S.Theocharis  | Add input ix Changed ix_UpstreamRunning
	 30/03/2020 | 3.3       | K.Pokorski    | Changed error reset condition
	 02/04/2020 | 3.4       | S.Theocharis  | Changed check to downsteam
	 03/05/2023 | 4.0       | F.Baten       | PEC delay changed to distance 4.0 Release TIA 17.5
	 12/03/2024  | 4.1      | S. Nieswiec   | Small variable name changes according to current standard
	*)

	REGION 1 - Triggers

	    // Rising edge PEC Jam.
	    #R_TRIG_PECJam(CLK := #s_Status.Jam);

	END_REGION

	REGION 2 - Active function

	    // To activate the Jam monitoring, the jam displacement limit must be greater than zero.
	    #sx_Enable := #iUDT_PECConfiguration.JamDisplacementLimit > 0;

	END_REGION

	REGION 3 - Reset errors

	    // Reset Jam error and initialize Jam displacement counter, when reset signal occurs.
	    IF #iqUDT_ConveyorInterface.InternalErrorReset
	        AND (#iUDT_PECConfiguration.ResetWithPECBlocked
	        OR (NOT #iUDT_PECConfiguration.ResetWithPECBlocked
	        AND #sx_PECFiltered AND #ix_PECDownstream))
	        AND #s_Status.Jam
	    THEN
	        #si_AuxJamDisplacement := 0;
	        #s_Status.Jam := FALSE;
	    END_IF;

	END_REGION

	REGION 4 - Photo eye filters

	    // End OF section photo eye signal filter measurement
	    #PEC_OnOffDelay(ii_Displacement := #iqUDT_ConveyorInterface.Displacement,
	                    idi_OnDelayDistance := #iUDT_PECConfiguration.OnDelayDistance,
	                    idi_OffDelayDistance := #iUDT_PECConfiguration.OffDelayDistance,
	                    ix_SignalToDelay := #ix_PEC,
	                    ix_Enable := TRUE,
	                    qx_DelayedSignal => #sx_PECFiltered);

	    // Write the current status of the photo eye.
	    #s_Status.PEC := #sx_PECFiltered;
	    #qx_PECFiltered := #sx_PECFiltered;

	END_REGION

	REGION 5 - Jam detection

	    // Increasing Jam displacement counter by conveyor displacement, when photo eyes on conveyor and downstream conveyor are blocked and jam functionality is enable.
	    IF #ix_PECDownstream AND (NOT #sx_PECFiltered) AND #sx_Enable AND #ix_DownstreamRunning

	    THEN
	        #si_AuxJamDisplacement += #iqUDT_ConveyorInterface.Displacement;
	    ELSE
	        #si_AuxJamDisplacement := 0;
	    END_IF;

	    // Set jam error when total jam displacement exceeded limit.
	    IF (#si_AuxJamDisplacement > #iUDT_PECConfiguration.JamDisplacementLimit)
	        OR (#si_AuxJamDisplacement < (#iUDT_PECConfiguration.JamDisplacementLimit * -1))
	    THEN
	        #s_Status.Jam := TRUE;
	    END_IF;

	END_REGION

	REGION 6 - Statistics

	    // Jam Photo eye blocked statistics.
	    IF #s_Status.Jam
	        OR #iqUDT_ConveyorInterface.ResetStatistics
	    THEN
	        "FC_Statistics"(ix_Reset := #iqUDT_ConveyorInterface.ResetStatistics,
	                        ix_Activate := #s_Status.Jam,
	                        ix_RTrigActivate := #R_TRIG_PECJam.Q,
	                        iqUDT_Statistics := #iqUDT_PECStatistics.Jam);
	    END_IF;

	END_REGION

	REGION 7 - Internal PEC error

	    // Set Internal photo eye error .
	    IF #s_Status.Jam
	    THEN
	        #iqUDT_ConveyorInterface.InternalErrorPEC := TRUE;
	    END_IF;

	END_REGION

	REGION 8 - Status

	    // Status update on change.
	    IF #s_StatusOld <> #s_Status
	    THEN
	        #qUDT_HMIStatus := #s_Status;
	        #s_StatusOld := #s_Status;
	    END_IF;

	END_REGION
END_FUNCTION_BLOCK

FUNCTION_BLOCK "FB_VfdSEWMOVI-CPositioning"
TITLE = FB_VFD_SEW_MOVI-C_Positioning
{ S7_Optimized_Access := 'TRUE' }
AUTHOR : MHSE
VERSION : 3.0
// ATTRIBUTES
// AUTO_NUMBER = True
// BLOCK_NUMBER = 36
// END_ATTRIBUTES
//Control SEW Servo VFD with multiple positions
   VAR_INPUT
      iUDT_VfdConfig { ExternalAccessible := 'False'; ExternalVisible := 'False'; ExternalWritable := 'False'} : "UDT_VfdPositioningConfiguration";   //  Configuration structure
      iUDT_VfdInputs { ExternalAccessible := 'False'; ExternalVisible := 'False'; ExternalWritable := 'False'} : "UDT_VfdSEWPositioningPI";   //  VFD inputs structure
      ix_MainPowerOk { ExternalAccessible := 'False'; ExternalVisible := 'False'; ExternalWritable := 'False'} : Bool;   //  True = Main power is ok
      ix_BackupPowerOk { ExternalAccessible := 'False'; ExternalVisible := 'False'; ExternalWritable := 'False'} : Bool;   //  True = back-up power is ok
      ix_SimulationModeActive { ExternalAccessible := 'False'; ExternalVisible := 'False'; ExternalWritable := 'False'} : Bool;   //  Simulation On
   END_VAR

   VAR_OUTPUT
      qUDT_HMIStatus { ExternalAccessible := 'False'; ExternalVisible := 'False'; ExternalWritable := 'False'} : "UDT_VfdPositioningStatus";   //  HMI status structure
      qUDT_VfdOutputs { ExternalAccessible := 'False'; ExternalVisible := 'False'; ExternalWritable := 'False'} : "UDT_VfdSEWPositioningPO";   //  VFD outputs structure
   END_VAR

   VAR_IN_OUT
      iqUDT_VSUInterface : "UDT_VSUInterface";   //  VSU interface structure
      iqUDT_VFDStatistics : "UDT_VfdStatistics";   //  VFD statistics
   END_VAR

